REGION Network 4: AV-20.04
   RUNG wire#powerrail
      #"AV-20.04"(FB_OPEN := wire#w1, FB_CLOSE := wire#w2, LOCK := #lock, ERR_EXTERN :=, LIOP_SEL := #Init, L_AUT := #Init, L_REMOTE := #Init, L_SIM :=, L_RESET := #Reset, AUT_OP :=, MAN_OP :=, SIM_OP :=, L_MON := #Init, MON_T :=, MON_T_CLOSE :=, INSTANCE := 'AV-20.04', RESTART :=, VISIBILITY :=, OPdwCmd :=, QdwState =>, QwState =>, QCLOSING =>, QCLOSE =>, QOPENING =>, QOPEN =>, QCMD_OP => "AV-20.04", QMON =>, QMON_ERR =>, QMON_T =>, QMON_T_CLOSE =>, QMAN_AUT =>, QREMOTE =>, QSIM =>, QLOCK =>, QERR =>, QERR_EXT =>, QwAlarm =>)
   END_RUNG
   RUNG wire#powerrail
      Contact( #"AV-20.04".QCMD_OP )
   END_RUNG wire#w1
   RUNG wire#powerrail
      I_Contact( #"AV-20.04".QCMD_OP )
   END_RUNG wire#w2
   // the same network as SCL:
   #"AV-20.04"(LOCK := #lock,   // "Valve"
               LIOP_SEL := #Init,
               L_AUT := #Init,
               L_REMOTE := #Init,
               L_RESET := #Reset,
               FB_OPEN := #"AV-20.04".QCMD_OP,
               FB_CLOSE := NOT #"AV-20.04".QCMD_OP,
               L_MON := #Init,
               INSTANCE := 'AV-20.04',
               QCMD_OP => "AV-20.04");
END_REGION

REGION Network 5: AV-20.05
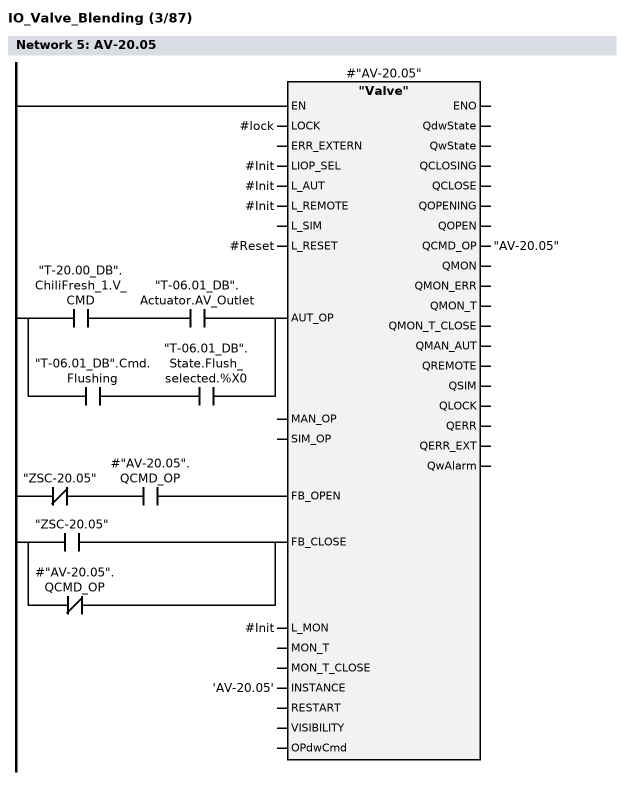
   RUNG wire#powerrail
      #"AV-20.05"(AUT_OP := wire#w1, FB_OPEN := wire#w2, FB_CLOSE := wire#w3, LOCK := #lock, ERR_EXTERN :=, LIOP_SEL := #Init, L_AUT := #Init, L_REMOTE := #Init, L_SIM :=, L_RESET := #Reset, MAN_OP :=, SIM_OP :=, L_MON := #Init, MON_T :=, MON_T_CLOSE :=, INSTANCE := 'AV-20.05', RESTART :=, VISIBILITY :=, OPdwCmd :=, QdwState =>, QwState =>, QCLOSING =>, QCLOSE =>, QOPENING =>, QOPEN =>, QCMD_OP => "AV-20.05", QMON =>, QMON_ERR =>, QMON_T =>, QMON_T_CLOSE =>, QMAN_AUT =>, QREMOTE =>, QSIM =>, QLOCK =>, QERR =>, QERR_EXT =>, QwAlarm =>)
   END_RUNG
   RUNG wire#powerrail
      Contact( "T-20.00_DB".ChiliFresh_1.V_CMD )
      Contact( "T-06.01_DB".Actuator.AV_Outlet )
   END_RUNG wire#w1
   RUNG wire#powerrail
      Contact( "T-06.01_DB".Cmd.Flushing )
      Contact( "T-06.01_DB".State.Flush_selected.%X0 )
   END_RUNG wire#w1
   RUNG wire#powerrail
      I_Contact( "ZSC-20.05" )
      Contact( #"AV-20.05".QCMD_OP )
   END_RUNG wire#w2
   RUNG wire#powerrail
      Contact( "ZSC-20.05" )
   END_RUNG wire#w3
   RUNG wire#powerrail
      I_Contact( #"AV-20.05".QCMD_OP )
   END_RUNG wire#w3
   // the same network as SCL:
   #"AV-20.05"(LOCK := #lock,   // "Valve"
               LIOP_SEL := #Init,
               L_AUT := #Init,
               L_REMOTE := #Init,
               L_RESET := #Reset,
               AUT_OP := ("T-20.00_DB".ChiliFresh_1.V_CMD AND "T-06.01_DB".Actuator.AV_Outlet) OR ("T-06.01_DB".Cmd.Flushing AND "T-06.01_DB".State.Flush_selected.%X0),
               FB_OPEN := NOT "ZSC-20.05" AND #"AV-20.05".QCMD_OP,
               FB_CLOSE := "ZSC-20.05" OR NOT #"AV-20.05".QCMD_OP,
               L_MON := #Init,
               INSTANCE := 'AV-20.05',
               QCMD_OP => "AV-20.05");
END_REGION

REGION Network 6: AV-20.06
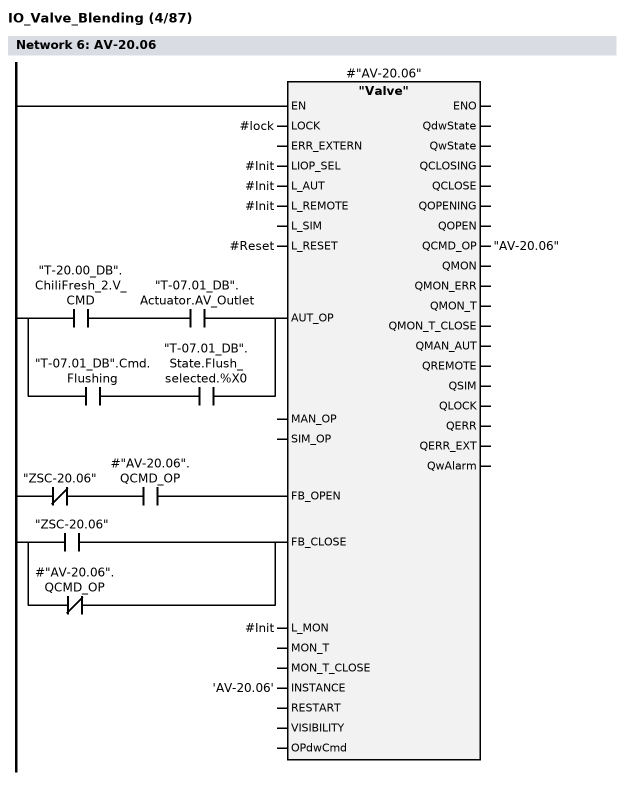
   RUNG wire#powerrail
      #"AV-20.06"(AUT_OP := wire#w1, FB_OPEN := wire#w2, FB_CLOSE := wire#w3, LOCK := #lock, ERR_EXTERN :=, LIOP_SEL := #Init, L_AUT := #Init, L_REMOTE := #Init, L_SIM :=, L_RESET := #Reset, MAN_OP :=, SIM_OP :=, L_MON := #Init, MON_T :=, MON_T_CLOSE :=, INSTANCE := 'AV-20.06', RESTART :=, VISIBILITY :=, OPdwCmd :=, QdwState =>, QwState =>, QCLOSING =>, QCLOSE =>, QOPENING =>, QOPEN =>, QCMD_OP => "AV-20.06", QMON =>, QMON_ERR =>, QMON_T =>, QMON_T_CLOSE =>, QMAN_AUT =>, QREMOTE =>, QSIM =>, QLOCK =>, QERR =>, QERR_EXT =>, QwAlarm =>)
   END_RUNG
   RUNG wire#powerrail
      Contact( "T-20.00_DB".ChiliFresh_2.V_CMD )
      Contact( "T-07.01_DB".Actuator.AV_Outlet )
   END_RUNG wire#w1
   RUNG wire#powerrail
      Contact( "T-07.01_DB".Cmd.Flushing )
      Contact( "T-07.01_DB".State.Flush_selected.%X0 )
   END_RUNG wire#w1
   RUNG wire#powerrail
      I_Contact( "ZSC-20.06" )
      Contact( #"AV-20.06".QCMD_OP )
   END_RUNG wire#w2
   RUNG wire#powerrail
      Contact( "ZSC-20.06" )
   END_RUNG wire#w3
   RUNG wire#powerrail
      I_Contact( #"AV-20.06".QCMD_OP )
   END_RUNG wire#w3
   // the same network as SCL:
   #"AV-20.06"(LOCK := #lock,   // "Valve"
               LIOP_SEL := #Init,
               L_AUT := #Init,
               L_REMOTE := #Init,
               L_RESET := #Reset,
               AUT_OP := ("T-20.00_DB".ChiliFresh_2.V_CMD AND "T-07.01_DB".Actuator.AV_Outlet) OR ("T-07.01_DB".Cmd.Flushing AND "T-07.01_DB".State.Flush_selected.%X0),
               FB_OPEN := NOT "ZSC-20.06" AND #"AV-20.06".QCMD_OP,
               FB_CLOSE := "ZSC-20.06" OR NOT #"AV-20.06".QCMD_OP,
               L_MON := #Init,
               INSTANCE := 'AV-20.06',
               QCMD_OP => "AV-20.06");
END_REGION

REGION Network 7: AV-20.07
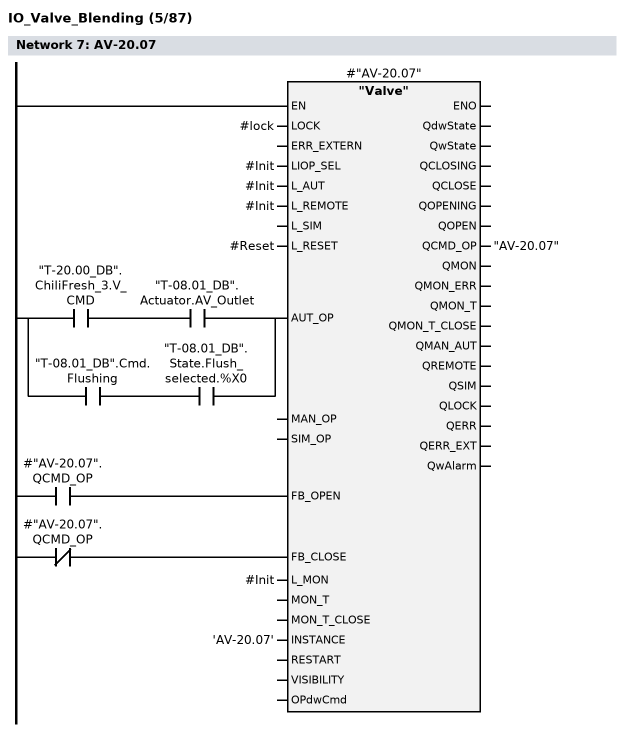
   RUNG wire#powerrail
      #"AV-20.07"(AUT_OP := wire#w1, FB_OPEN := wire#w2, FB_CLOSE := wire#w3, LOCK := #lock, ERR_EXTERN :=, LIOP_SEL := #Init, L_AUT := #Init, L_REMOTE := #Init, L_SIM :=, L_RESET := #Reset, MAN_OP :=, SIM_OP :=, L_MON := #Init, MON_T :=, MON_T_CLOSE :=, INSTANCE := 'AV-20.07', RESTART :=, VISIBILITY :=, OPdwCmd :=, QdwState =>, QwState =>, QCLOSING =>, QCLOSE =>, QOPENING =>, QOPEN =>, QCMD_OP => "AV-20.07", QMON =>, QMON_ERR =>, QMON_T =>, QMON_T_CLOSE =>, QMAN_AUT =>, QREMOTE =>, QSIM =>, QLOCK =>, QERR =>, QERR_EXT =>, QwAlarm =>)
   END_RUNG
   RUNG wire#powerrail
      Contact( "T-20.00_DB".ChiliFresh_3.V_CMD )
      Contact( "T-08.01_DB".Actuator.AV_Outlet )
   END_RUNG wire#w1
   RUNG wire#powerrail
      Contact( "T-08.01_DB".Cmd.Flushing )
      Contact( "T-08.01_DB".State.Flush_selected.%X0 )
   END_RUNG wire#w1
   RUNG wire#powerrail
      Contact( #"AV-20.07".QCMD_OP )
   END_RUNG wire#w2
   RUNG wire#powerrail
      I_Contact( #"AV-20.07".QCMD_OP )
   END_RUNG wire#w3
   // the same network as SCL:
   #"AV-20.07"(LOCK := #lock,   // "Valve"
               LIOP_SEL := #Init,
               L_AUT := #Init,
               L_REMOTE := #Init,
               L_RESET := #Reset,
               AUT_OP := ("T-20.00_DB".ChiliFresh_3.V_CMD AND "T-08.01_DB".Actuator.AV_Outlet) OR ("T-08.01_DB".Cmd.Flushing AND "T-08.01_DB".State.Flush_selected.%X0),
               FB_OPEN := #"AV-20.07".QCMD_OP,
               FB_CLOSE := NOT #"AV-20.07".QCMD_OP,
               L_MON := #Init,
               INSTANCE := 'AV-20.07',
               QCMD_OP => "AV-20.07");
END_REGION

REGION Network 8: AV-20.08
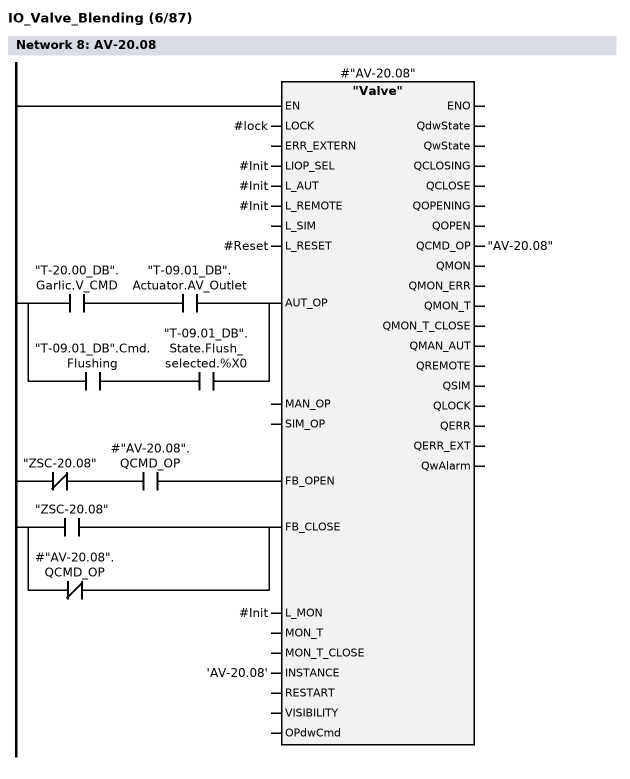
   RUNG wire#powerrail
      #"AV-20.08"(AUT_OP := wire#w1, FB_OPEN := wire#w2, FB_CLOSE := wire#w3, LOCK := #lock, ERR_EXTERN :=, LIOP_SEL := #Init, L_AUT := #Init, L_REMOTE := #Init, L_SIM :=, L_RESET := #Reset, MAN_OP :=, SIM_OP :=, L_MON := #Init, MON_T :=, MON_T_CLOSE :=, INSTANCE := 'AV-20.08', RESTART :=, VISIBILITY :=, OPdwCmd :=, QdwState =>, QwState =>, QCLOSING =>, QCLOSE =>, QOPENING =>, QOPEN =>, QCMD_OP => "AV-20.08", QMON =>, QMON_ERR =>, QMON_T =>, QMON_T_CLOSE =>, QMAN_AUT =>, QREMOTE =>, QSIM =>, QLOCK =>, QERR =>, QERR_EXT =>, QwAlarm =>)
   END_RUNG
   RUNG wire#powerrail
      Contact( "T-20.00_DB".Garlic.V_CMD )
      Contact( "T-09.01_DB".Actuator.AV_Outlet )
   END_RUNG wire#w1
   RUNG wire#powerrail
      Contact( "T-09.01_DB".Cmd.Flushing )
      Contact( "T-09.01_DB".State.Flush_selected.%X0 )
   END_RUNG wire#w1
   RUNG wire#powerrail
      I_Contact( "ZSC-20.08" )
      Contact( #"AV-20.08".QCMD_OP )
   END_RUNG wire#w2
   RUNG wire#powerrail
      Contact( "ZSC-20.08" )
   END_RUNG wire#w3
   RUNG wire#powerrail
      I_Contact( #"AV-20.08".QCMD_OP )
   END_RUNG wire#w3
   // the same network as SCL:
   #"AV-20.08"(LOCK := #lock,   // "Valve"
               LIOP_SEL := #Init,
               L_AUT := #Init,
               L_REMOTE := #Init,
               L_RESET := #Reset,
               AUT_OP := ("T-20.00_DB".Garlic.V_CMD AND "T-09.01_DB".Actuator.AV_Outlet) OR ("T-09.01_DB".Cmd.Flushing AND "T-09.01_DB".State.Flush_selected.%X0),
               FB_OPEN := NOT "ZSC-20.08" AND #"AV-20.08".QCMD_OP,
               FB_CLOSE := "ZSC-20.08" OR NOT #"AV-20.08".QCMD_OP,
               L_MON := #Init,
               INSTANCE := 'AV-20.08',
               QCMD_OP => "AV-20.08");
END_REGION

REGION Network 9: AV-20.09
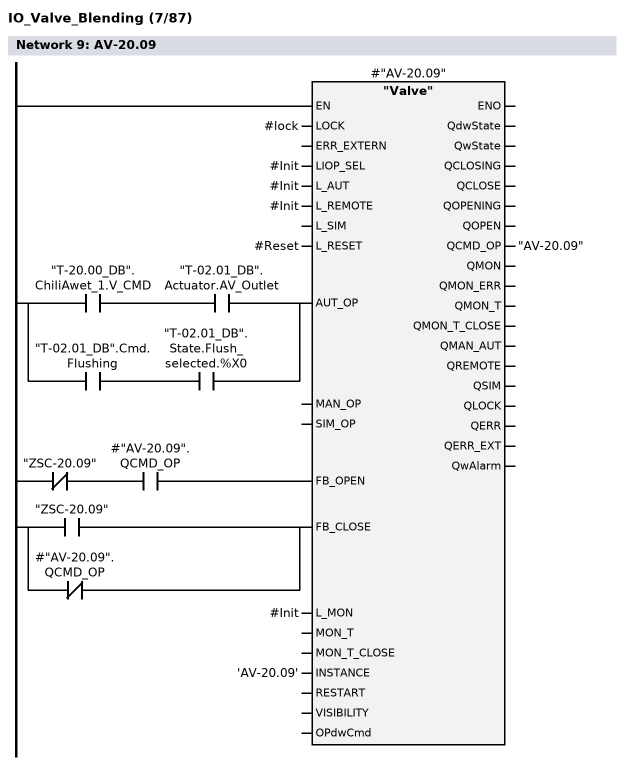
   RUNG wire#powerrail
      #"AV-20.09"(AUT_OP := wire#w1, FB_OPEN := wire#w2, FB_CLOSE := wire#w3, LOCK := #lock, ERR_EXTERN :=, LIOP_SEL := #Init, L_AUT := #Init, L_REMOTE := #Init, L_SIM :=, L_RESET := #Reset, MAN_OP :=, SIM_OP :=, L_MON := #Init, MON_T :=, MON_T_CLOSE :=, INSTANCE := 'AV-20.09', RESTART :=, VISIBILITY :=, OPdwCmd :=, QdwState =>, QwState =>, QCLOSING =>, QCLOSE =>, QOPENING =>, QOPEN =>, QCMD_OP => "AV-20.09", QMON =>, QMON_ERR =>, QMON_T =>, QMON_T_CLOSE =>, QMAN_AUT =>, QREMOTE =>, QSIM =>, QLOCK =>, QERR =>, QERR_EXT =>, QwAlarm =>)
   END_RUNG
   RUNG wire#powerrail
      Contact( "T-20.00_DB".ChiliAwet_1.V_CMD )
      Contact( "T-02.01_DB".Actuator.AV_Outlet )
   END_RUNG wire#w1
   RUNG wire#powerrail
      Contact( "T-02.01_DB".Cmd.Flushing )
      Contact( "T-02.01_DB".State.Flush_selected.%X0 )
   END_RUNG wire#w1
   RUNG wire#powerrail
      I_Contact( "ZSC-20.09" )
      Contact( #"AV-20.09".QCMD_OP )
   END_RUNG wire#w2
   RUNG wire#powerrail
      Contact( "ZSC-20.09" )
   END_RUNG wire#w3
   RUNG wire#powerrail
      I_Contact( #"AV-20.09".QCMD_OP )
   END_RUNG wire#w3
   // the same network as SCL:
   #"AV-20.09"(LOCK := #lock,   // "Valve"
               LIOP_SEL := #Init,
               L_AUT := #Init,
               L_REMOTE := #Init,
               L_RESET := #Reset,
               AUT_OP := ("T-20.00_DB".ChiliAwet_1.V_CMD AND "T-02.01_DB".Actuator.AV_Outlet) OR ("T-02.01_DB".Cmd.Flushing AND "T-02.01_DB".State.Flush_selected.%X0),
               FB_OPEN := NOT "ZSC-20.09" AND #"AV-20.09".QCMD_OP,
               FB_CLOSE := "ZSC-20.09" OR NOT #"AV-20.09".QCMD_OP,
               L_MON := #Init,
               INSTANCE := 'AV-20.09',
               QCMD_OP => "AV-20.09");
END_REGION

REGION Network 10: AV-20.10
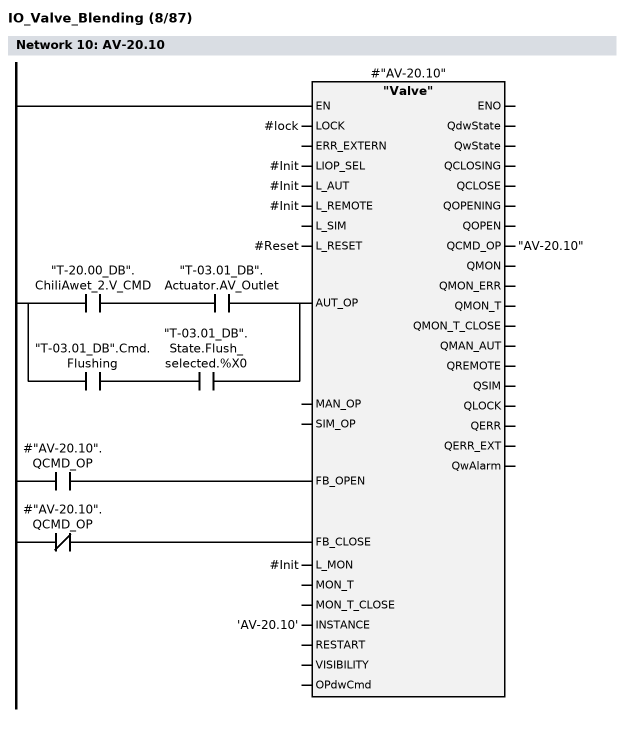
   RUNG wire#powerrail
      #"AV-20.10"(AUT_OP := wire#w1, FB_OPEN := wire#w2, FB_CLOSE := wire#w3, LOCK := #lock, ERR_EXTERN :=, LIOP_SEL := #Init, L_AUT := #Init, L_REMOTE := #Init, L_SIM :=, L_RESET := #Reset, MAN_OP :=, SIM_OP :=, L_MON := #Init, MON_T :=, MON_T_CLOSE :=, INSTANCE := 'AV-20.10', RESTART :=, VISIBILITY :=, OPdwCmd :=, QdwState =>, QwState =>, QCLOSING =>, QCLOSE =>, QOPENING =>, QOPEN =>, QCMD_OP => "AV-20.10", QMON =>, QMON_ERR =>, QMON_T =>, QMON_T_CLOSE =>, QMAN_AUT =>, QREMOTE =>, QSIM =>, QLOCK =>, QERR =>, QERR_EXT =>, QwAlarm =>)
   END_RUNG
   RUNG wire#powerrail
      Contact( "T-20.00_DB".ChiliAwet_2.V_CMD )
      Contact( "T-03.01_DB".Actuator.AV_Outlet )
   END_RUNG wire#w1
   RUNG wire#powerrail
      Contact( "T-03.01_DB".Cmd.Flushing )
      Contact( "T-03.01_DB".State.Flush_selected.%X0 )
   END_RUNG wire#w1
   RUNG wire#powerrail
      Contact( #"AV-20.10".QCMD_OP )
   END_RUNG wire#w2
   RUNG wire#powerrail
      I_Contact( #"AV-20.10".QCMD_OP )
   END_RUNG wire#w3
   // the same network as SCL:
   #"AV-20.10"(LOCK := #lock,   // "Valve"
               LIOP_SEL := #Init,
               L_AUT := #Init,
               L_REMOTE := #Init,
               L_RESET := #Reset,
               AUT_OP := ("T-20.00_DB".ChiliAwet_2.V_CMD AND "T-03.01_DB".Actuator.AV_Outlet) OR ("T-03.01_DB".Cmd.Flushing AND "T-03.01_DB".State.Flush_selected.%X0),
               FB_OPEN := #"AV-20.10".QCMD_OP,
               FB_CLOSE := NOT #"AV-20.10".QCMD_OP,
               L_MON := #Init,
               INSTANCE := 'AV-20.10',
               QCMD_OP => "AV-20.10");
END_REGION

REGION Network 11: AV-20.11
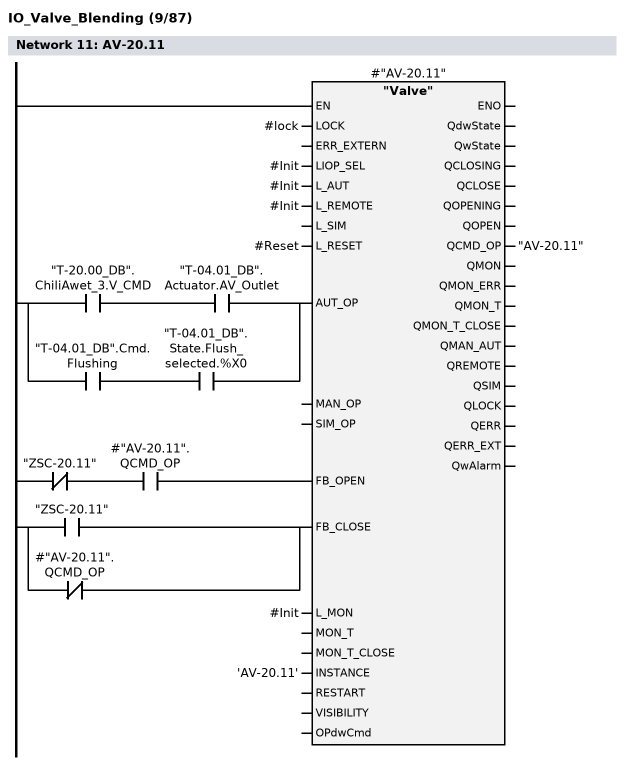
   RUNG wire#powerrail
      #"AV-20.11"(AUT_OP := wire#w1, FB_OPEN := wire#w2, FB_CLOSE := wire#w3, LOCK := #lock, ERR_EXTERN :=, LIOP_SEL := #Init, L_AUT := #Init, L_REMOTE := #Init, L_SIM :=, L_RESET := #Reset, MAN_OP :=, SIM_OP :=, L_MON := #Init, MON_T :=, MON_T_CLOSE :=, INSTANCE := 'AV-20.11', RESTART :=, VISIBILITY :=, OPdwCmd :=, QdwState =>, QwState =>, QCLOSING =>, QCLOSE =>, QOPENING =>, QOPEN =>, QCMD_OP => "AV-20.11", QMON =>, QMON_ERR =>, QMON_T =>, QMON_T_CLOSE =>, QMAN_AUT =>, QREMOTE =>, QSIM =>, QLOCK =>, QERR =>, QERR_EXT =>, QwAlarm =>)
   END_RUNG
   RUNG wire#powerrail
      Contact( "T-20.00_DB".ChiliAwet_3.V_CMD )
      Contact( "T-04.01_DB".Actuator.AV_Outlet )
   END_RUNG wire#w1
   RUNG wire#powerrail
      Contact( "T-04.01_DB".Cmd.Flushing )
      Contact( "T-04.01_DB".State.Flush_selected.%X0 )
   END_RUNG wire#w1
   RUNG wire#powerrail
      I_Contact( "ZSC-20.11" )
      Contact( #"AV-20.11".QCMD_OP )
   END_RUNG wire#w2
   RUNG wire#powerrail
      Contact( "ZSC-20.11" )
   END_RUNG wire#w3
   RUNG wire#powerrail
      I_Contact( #"AV-20.11".QCMD_OP )
   END_RUNG wire#w3
   // the same network as SCL:
   #"AV-20.11"(LOCK := #lock,   // "Valve"
               LIOP_SEL := #Init,
               L_AUT := #Init,
               L_REMOTE := #Init,
               L_RESET := #Reset,
               AUT_OP := ("T-20.00_DB".ChiliAwet_3.V_CMD AND "T-04.01_DB".Actuator.AV_Outlet) OR ("T-04.01_DB".Cmd.Flushing AND "T-04.01_DB".State.Flush_selected.%X0),
               FB_OPEN := NOT "ZSC-20.11" AND #"AV-20.11".QCMD_OP,
               FB_CLOSE := "ZSC-20.11" OR NOT #"AV-20.11".QCMD_OP,
               L_MON := #Init,
               INSTANCE := 'AV-20.11',
               QCMD_OP => "AV-20.11");
END_REGION

REGION Network 12: AV-20.12
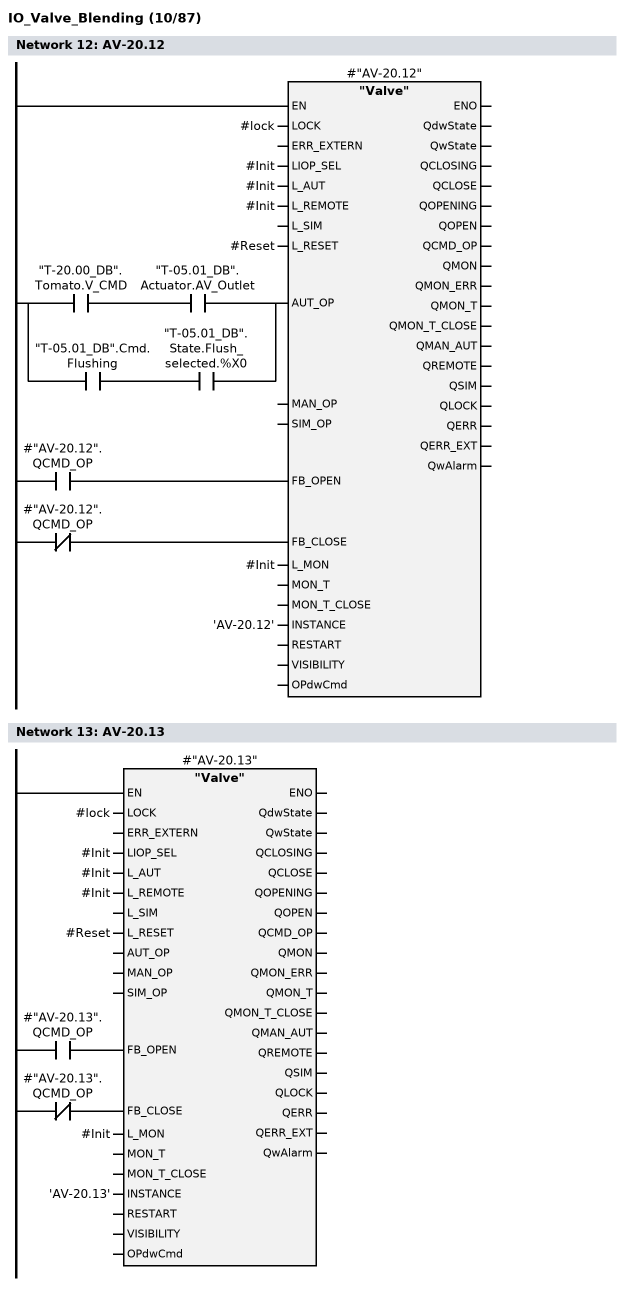
   RUNG wire#powerrail
      #"AV-20.12"(AUT_OP := wire#w1, FB_OPEN := wire#w2, FB_CLOSE := wire#w3, LOCK := #lock, ERR_EXTERN :=, LIOP_SEL := #Init, L_AUT := #Init, L_REMOTE := #Init, L_SIM :=, L_RESET := #Reset, MAN_OP :=, SIM_OP :=, L_MON := #Init, MON_T :=, MON_T_CLOSE :=, INSTANCE := 'AV-20.12', RESTART :=, VISIBILITY :=, OPdwCmd :=, QdwState =>, QwState =>, QCLOSING =>, QCLOSE =>, QOPENING =>, QOPEN =>, QCMD_OP =>, QMON =>, QMON_ERR =>, QMON_T =>, QMON_T_CLOSE =>, QMAN_AUT =>, QREMOTE =>, QSIM =>, QLOCK =>, QERR =>, QERR_EXT =>, QwAlarm =>)
   END_RUNG
   RUNG wire#powerrail
      Contact( "T-20.00_DB".Tomato.V_CMD )
      Contact( "T-05.01_DB".Actuator.AV_Outlet )
   END_RUNG wire#w1
   RUNG wire#powerrail
      Contact( "T-05.01_DB".Cmd.Flushing )
      Contact( "T-05.01_DB".State.Flush_selected.%X0 )
   END_RUNG wire#w1
   RUNG wire#powerrail
      Contact( #"AV-20.12".QCMD_OP )
   END_RUNG wire#w2
   RUNG wire#powerrail
      I_Contact( #"AV-20.12".QCMD_OP )
   END_RUNG wire#w3
   // the same network as SCL:
   #"AV-20.12"(LOCK := #lock,   // "Valve"
               LIOP_SEL := #Init,
               L_AUT := #Init,
               L_REMOTE := #Init,
               L_RESET := #Reset,
               AUT_OP := ("T-20.00_DB".Tomato.V_CMD AND "T-05.01_DB".Actuator.AV_Outlet) OR ("T-05.01_DB".Cmd.Flushing AND "T-05.01_DB".State.Flush_selected.%X0),
               FB_OPEN := #"AV-20.12".QCMD_OP,
               FB_CLOSE := NOT #"AV-20.12".QCMD_OP,
               L_MON := #Init,
               INSTANCE := 'AV-20.12');
END_REGION

REGION Network 13: AV-20.13
   RUNG wire#powerrail
      #"AV-20.13"(FB_OPEN := wire#w1, FB_CLOSE := wire#w2, LOCK := #lock, ERR_EXTERN :=, LIOP_SEL := #Init, L_AUT := #Init, L_REMOTE := #Init, L_SIM :=, L_RESET := #Reset, AUT_OP :=, MAN_OP :=, SIM_OP :=, L_MON := #Init, MON_T :=, MON_T_CLOSE :=, INSTANCE := 'AV-20.13', RESTART :=, VISIBILITY :=, OPdwCmd :=, QdwState =>, QwState =>, QCLOSING =>, QCLOSE =>, QOPENING =>, QOPEN =>, QCMD_OP =>, QMON =>, QMON_ERR =>, QMON_T =>, QMON_T_CLOSE =>, QMAN_AUT =>, QREMOTE =>, QSIM =>, QLOCK =>, QERR =>, QERR_EXT =>, QwAlarm =>)
   END_RUNG
   RUNG wire#powerrail
      Contact( #"AV-20.13".QCMD_OP )
   END_RUNG wire#w1
   RUNG wire#powerrail
      I_Contact( #"AV-20.13".QCMD_OP )
   END_RUNG wire#w2
   // the same network as SCL:
   #"AV-20.13"(LOCK := #lock,   // "Valve"
               LIOP_SEL := #Init,
               L_AUT := #Init,
               L_REMOTE := #Init,
               L_RESET := #Reset,
               FB_OPEN := #"AV-20.13".QCMD_OP,
               FB_CLOSE := NOT #"AV-20.13".QCMD_OP,
               L_MON := #Init,
               INSTANCE := 'AV-20.13');
END_REGION

REGION Network 14: AV-20.14
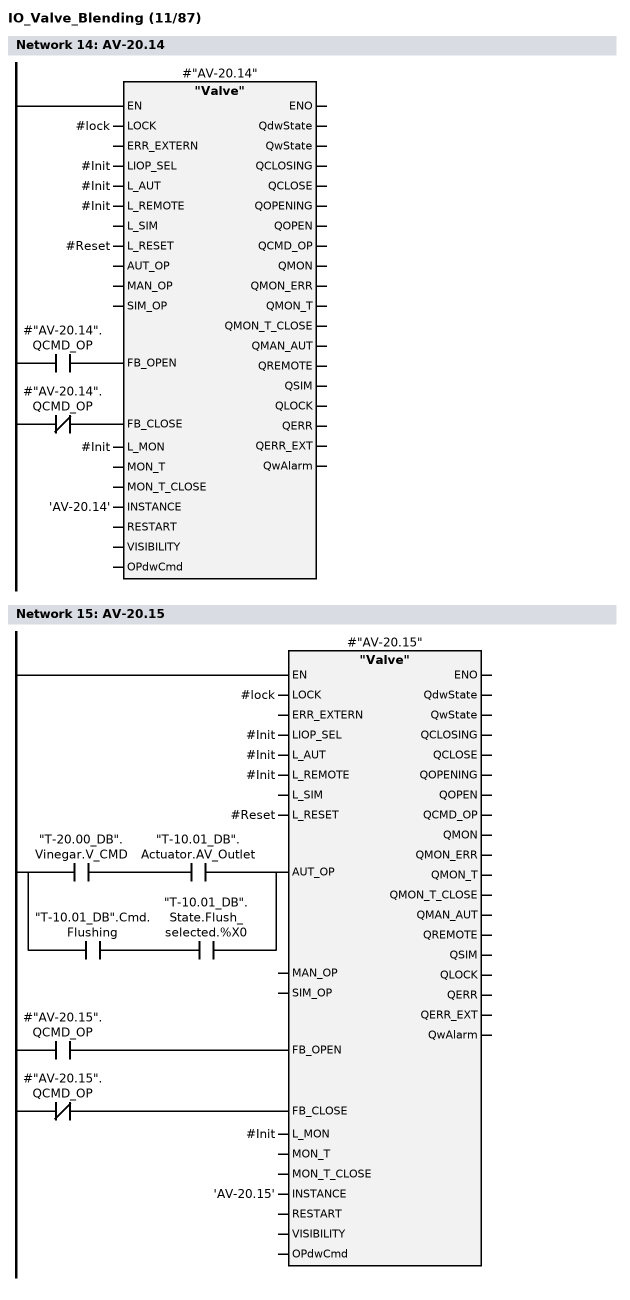
   RUNG wire#powerrail
      #"AV-20.14"(FB_OPEN := wire#w1, FB_CLOSE := wire#w2, LOCK := #lock, ERR_EXTERN :=, LIOP_SEL := #Init, L_AUT := #Init, L_REMOTE := #Init, L_SIM :=, L_RESET := #Reset, AUT_OP :=, MAN_OP :=, SIM_OP :=, L_MON := #Init, MON_T :=, MON_T_CLOSE :=, INSTANCE := 'AV-20.14', RESTART :=, VISIBILITY :=, OPdwCmd :=, QdwState =>, QwState =>, QCLOSING =>, QCLOSE =>, QOPENING =>, QOPEN =>, QCMD_OP =>, QMON =>, QMON_ERR =>, QMON_T =>, QMON_T_CLOSE =>, QMAN_AUT =>, QREMOTE =>, QSIM =>, QLOCK =>, QERR =>, QERR_EXT =>, QwAlarm =>)
   END_RUNG
   RUNG wire#powerrail
      Contact( #"AV-20.14".QCMD_OP )
   END_RUNG wire#w1
   RUNG wire#powerrail
      I_Contact( #"AV-20.14".QCMD_OP )
   END_RUNG wire#w2
   // the same network as SCL:
   #"AV-20.14"(LOCK := #lock,   // "Valve"
               LIOP_SEL := #Init,
               L_AUT := #Init,
               L_REMOTE := #Init,
               L_RESET := #Reset,
               FB_OPEN := #"AV-20.14".QCMD_OP,
               FB_CLOSE := NOT #"AV-20.14".QCMD_OP,
               L_MON := #Init,
               INSTANCE := 'AV-20.14');
END_REGION

REGION Network 15: AV-20.15
   RUNG wire#powerrail
      #"AV-20.15"(AUT_OP := wire#w1, FB_OPEN := wire#w2, FB_CLOSE := wire#w3, LOCK := #lock, ERR_EXTERN :=, LIOP_SEL := #Init, L_AUT := #Init, L_REMOTE := #Init, L_SIM :=, L_RESET := #Reset, MAN_OP :=, SIM_OP :=, L_MON := #Init, MON_T :=, MON_T_CLOSE :=, INSTANCE := 'AV-20.15', RESTART :=, VISIBILITY :=, OPdwCmd :=, QdwState =>, QwState =>, QCLOSING =>, QCLOSE =>, QOPENING =>, QOPEN =>, QCMD_OP =>, QMON =>, QMON_ERR =>, QMON_T =>, QMON_T_CLOSE =>, QMAN_AUT =>, QREMOTE =>, QSIM =>, QLOCK =>, QERR =>, QERR_EXT =>, QwAlarm =>)
   END_RUNG
   RUNG wire#powerrail
      Contact( "T-20.00_DB".Vinegar.V_CMD )
      Contact( "T-10.01_DB".Actuator.AV_Outlet )
   END_RUNG wire#w1
   RUNG wire#powerrail
      Contact( "T-10.01_DB".Cmd.Flushing )
      Contact( "T-10.01_DB".State.Flush_selected.%X0 )
   END_RUNG wire#w1
   RUNG wire#powerrail
      Contact( #"AV-20.15".QCMD_OP )
   END_RUNG wire#w2
   RUNG wire#powerrail
      I_Contact( #"AV-20.15".QCMD_OP )
   END_RUNG wire#w3
   // the same network as SCL:
   #"AV-20.15"(LOCK := #lock,   // "Valve"
               LIOP_SEL := #Init,
               L_AUT := #Init,
               L_REMOTE := #Init,
               L_RESET := #Reset,
               AUT_OP := ("T-20.00_DB".Vinegar.V_CMD AND "T-10.01_DB".Actuator.AV_Outlet) OR ("T-10.01_DB".Cmd.Flushing AND "T-10.01_DB".State.Flush_selected.%X0),
               FB_OPEN := #"AV-20.15".QCMD_OP,
               FB_CLOSE := NOT #"AV-20.15".QCMD_OP,
               L_MON := #Init,
               INSTANCE := 'AV-20.15');
END_REGION

REGION Network 16: AV-20.16
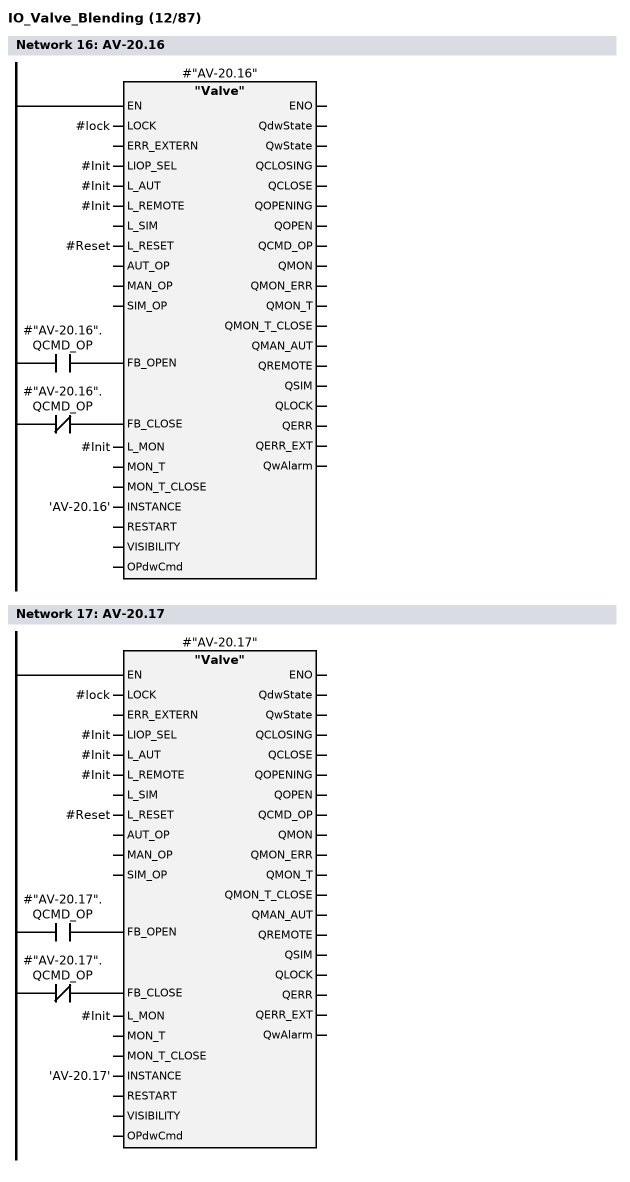
   RUNG wire#powerrail
      #"AV-20.16"(FB_OPEN := wire#w1, FB_CLOSE := wire#w2, LOCK := #lock, ERR_EXTERN :=, LIOP_SEL := #Init, L_AUT := #Init, L_REMOTE := #Init, L_SIM :=, L_RESET := #Reset, AUT_OP :=, MAN_OP :=, SIM_OP :=, L_MON := #Init, MON_T :=, MON_T_CLOSE :=, INSTANCE := 'AV-20.16', RESTART :=, VISIBILITY :=, OPdwCmd :=, QdwState =>, QwState =>, QCLOSING =>, QCLOSE =>, QOPENING =>, QOPEN =>, QCMD_OP =>, QMON =>, QMON_ERR =>, QMON_T =>, QMON_T_CLOSE =>, QMAN_AUT =>, QREMOTE =>, QSIM =>, QLOCK =>, QERR =>, QERR_EXT =>, QwAlarm =>)
   END_RUNG
   RUNG wire#powerrail
      Contact( #"AV-20.16".QCMD_OP )
   END_RUNG wire#w1
   RUNG wire#powerrail
      I_Contact( #"AV-20.16".QCMD_OP )
   END_RUNG wire#w2
   // the same network as SCL:
   #"AV-20.16"(LOCK := #lock,   // "Valve"
               LIOP_SEL := #Init,
               L_AUT := #Init,
               L_REMOTE := #Init,
               L_RESET := #Reset,
               FB_OPEN := #"AV-20.16".QCMD_OP,
               FB_CLOSE := NOT #"AV-20.16".QCMD_OP,
               L_MON := #Init,
               INSTANCE := 'AV-20.16');
END_REGION

REGION Network 17: AV-20.17
   RUNG wire#powerrail
      #"AV-20.17"(FB_OPEN := wire#w1, FB_CLOSE := wire#w2, LOCK := #lock, ERR_EXTERN :=, LIOP_SEL := #Init, L_AUT := #Init, L_REMOTE := #Init, L_SIM :=, L_RESET := #Reset, AUT_OP :=, MAN_OP :=, SIM_OP :=, L_MON := #Init, MON_T :=, MON_T_CLOSE :=, INSTANCE := 'AV-20.17', RESTART :=, VISIBILITY :=, OPdwCmd :=, QdwState =>, QwState =>, QCLOSING =>, QCLOSE =>, QOPENING =>, QOPEN =>, QCMD_OP =>, QMON =>, QMON_ERR =>, QMON_T =>, QMON_T_CLOSE =>, QMAN_AUT =>, QREMOTE =>, QSIM =>, QLOCK =>, QERR =>, QERR_EXT =>, QwAlarm =>)
   END_RUNG
   RUNG wire#powerrail
      Contact( #"AV-20.17".QCMD_OP )
   END_RUNG wire#w1
   RUNG wire#powerrail
      I_Contact( #"AV-20.17".QCMD_OP )
   END_RUNG wire#w2
   // the same network as SCL:
   #"AV-20.17"(LOCK := #lock,   // "Valve"
               LIOP_SEL := #Init,
               L_AUT := #Init,
               L_REMOTE := #Init,
               L_RESET := #Reset,
               FB_OPEN := #"AV-20.17".QCMD_OP,
               FB_CLOSE := NOT #"AV-20.17".QCMD_OP,
               L_MON := #Init,
               INSTANCE := 'AV-20.17');
END_REGION

REGION Network 18: AV-20.31
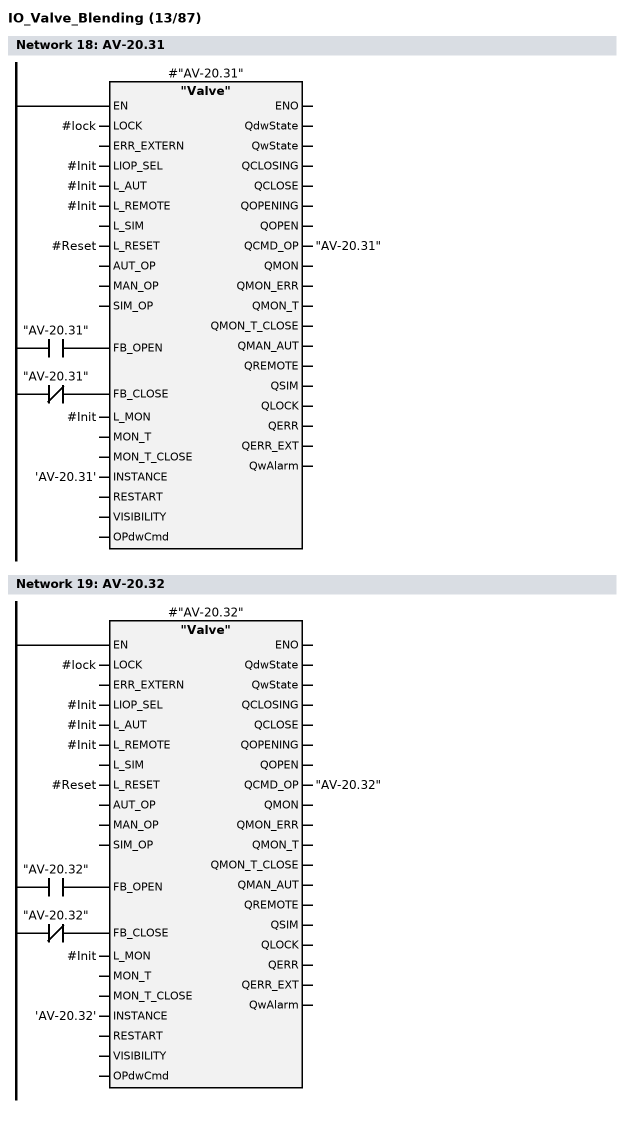
   RUNG wire#powerrail
      #"AV-20.31"(FB_OPEN := wire#w1, FB_CLOSE := wire#w2, LOCK := #lock, ERR_EXTERN :=, LIOP_SEL := #Init, L_AUT := #Init, L_REMOTE := #Init, L_SIM :=, L_RESET := #Reset, AUT_OP :=, MAN_OP :=, SIM_OP :=, L_MON := #Init, MON_T :=, MON_T_CLOSE :=, INSTANCE := 'AV-20.31', RESTART :=, VISIBILITY :=, OPdwCmd :=, QdwState =>, QwState =>, QCLOSING =>, QCLOSE =>, QOPENING =>, QOPEN =>, QCMD_OP => "AV-20.31", QMON =>, QMON_ERR =>, QMON_T =>, QMON_T_CLOSE =>, QMAN_AUT =>, QREMOTE =>, QSIM =>, QLOCK =>, QERR =>, QERR_EXT =>, QwAlarm =>)
   END_RUNG
   RUNG wire#powerrail
      Contact( "AV-20.31" )
   END_RUNG wire#w1
   RUNG wire#powerrail
      I_Contact( "AV-20.31" )
   END_RUNG wire#w2
   // the same network as SCL:
   #"AV-20.31"(LOCK := #lock,   // "Valve"
               LIOP_SEL := #Init,
               L_AUT := #Init,
               L_REMOTE := #Init,
               L_RESET := #Reset,
               FB_OPEN := "AV-20.31",
               FB_CLOSE := NOT "AV-20.31",
               L_MON := #Init,
               INSTANCE := 'AV-20.31',
               QCMD_OP => "AV-20.31");
END_REGION

REGION Network 19: AV-20.32
   RUNG wire#powerrail
      #"AV-20.32"(FB_OPEN := wire#w1, FB_CLOSE := wire#w2, LOCK := #lock, ERR_EXTERN :=, LIOP_SEL := #Init, L_AUT := #Init, L_REMOTE := #Init, L_SIM :=, L_RESET := #Reset, AUT_OP :=, MAN_OP :=, SIM_OP :=, L_MON := #Init, MON_T :=, MON_T_CLOSE :=, INSTANCE := 'AV-20.32', RESTART :=, VISIBILITY :=, OPdwCmd :=, QdwState =>, QwState =>, QCLOSING =>, QCLOSE =>, QOPENING =>, QOPEN =>, QCMD_OP => "AV-20.32", QMON =>, QMON_ERR =>, QMON_T =>, QMON_T_CLOSE =>, QMAN_AUT =>, QREMOTE =>, QSIM =>, QLOCK =>, QERR =>, QERR_EXT =>, QwAlarm =>)
   END_RUNG
   RUNG wire#powerrail
      Contact( "AV-20.32" )
   END_RUNG wire#w1
   RUNG wire#powerrail
      I_Contact( "AV-20.32" )
   END_RUNG wire#w2
   // the same network as SCL:
   #"AV-20.32"(LOCK := #lock,   // "Valve"
               LIOP_SEL := #Init,
               L_AUT := #Init,
               L_REMOTE := #Init,
               L_RESET := #Reset,
               FB_OPEN := "AV-20.32",
               FB_CLOSE := NOT "AV-20.32",
               L_MON := #Init,
               INSTANCE := 'AV-20.32',
               QCMD_OP => "AV-20.32");
END_REGION

REGION Network 20: AV-20.33
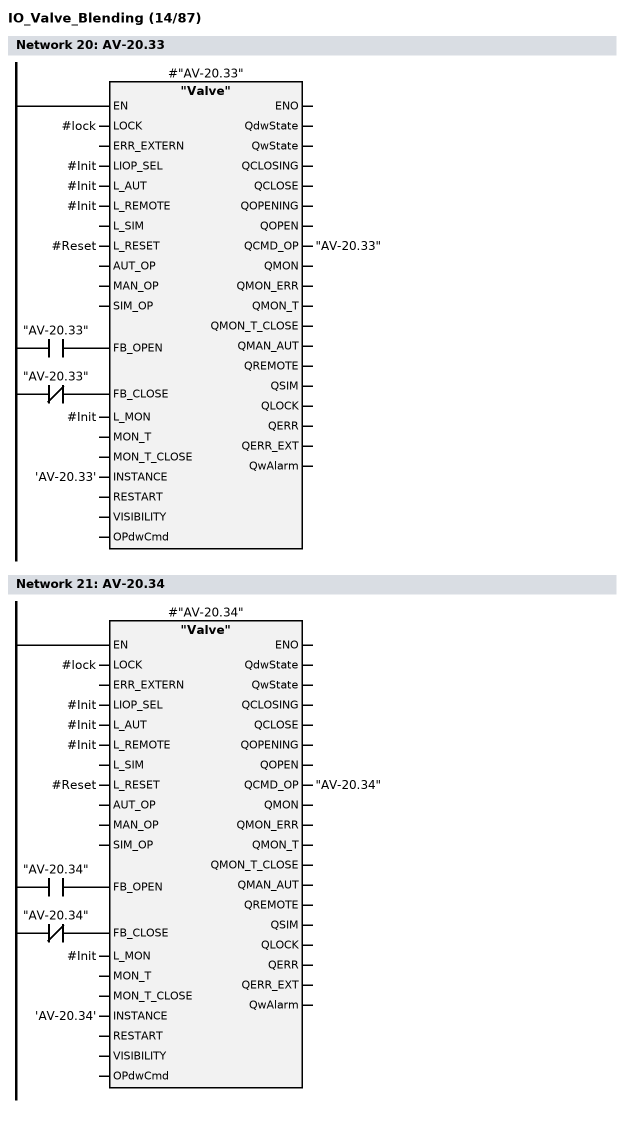
   RUNG wire#powerrail
      #"AV-20.33"(FB_OPEN := wire#w1, FB_CLOSE := wire#w2, LOCK := #lock, ERR_EXTERN :=, LIOP_SEL := #Init, L_AUT := #Init, L_REMOTE := #Init, L_SIM :=, L_RESET := #Reset, AUT_OP :=, MAN_OP :=, SIM_OP :=, L_MON := #Init, MON_T :=, MON_T_CLOSE :=, INSTANCE := 'AV-20.33', RESTART :=, VISIBILITY :=, OPdwCmd :=, QdwState =>, QwState =>, QCLOSING =>, QCLOSE =>, QOPENING =>, QOPEN =>, QCMD_OP => "AV-20.33", QMON =>, QMON_ERR =>, QMON_T =>, QMON_T_CLOSE =>, QMAN_AUT =>, QREMOTE =>, QSIM =>, QLOCK =>, QERR =>, QERR_EXT =>, QwAlarm =>)
   END_RUNG
   RUNG wire#powerrail
      Contact( "AV-20.33" )
   END_RUNG wire#w1
   RUNG wire#powerrail
      I_Contact( "AV-20.33" )
   END_RUNG wire#w2
   // the same network as SCL:
   #"AV-20.33"(LOCK := #lock,   // "Valve"
               LIOP_SEL := #Init,
               L_AUT := #Init,
               L_REMOTE := #Init,
               L_RESET := #Reset,
               FB_OPEN := "AV-20.33",
               FB_CLOSE := NOT "AV-20.33",
               L_MON := #Init,
               INSTANCE := 'AV-20.33',
               QCMD_OP => "AV-20.33");
END_REGION

REGION Network 21: AV-20.34
   RUNG wire#powerrail
      #"AV-20.34"(FB_OPEN := wire#w1, FB_CLOSE := wire#w2, LOCK := #lock, ERR_EXTERN :=, LIOP_SEL := #Init, L_AUT := #Init, L_REMOTE := #Init, L_SIM :=, L_RESET := #Reset, AUT_OP :=, MAN_OP :=, SIM_OP :=, L_MON := #Init, MON_T :=, MON_T_CLOSE :=, INSTANCE := 'AV-20.34', RESTART :=, VISIBILITY :=, OPdwCmd :=, QdwState =>, QwState =>, QCLOSING =>, QCLOSE =>, QOPENING =>, QOPEN =>, QCMD_OP => "AV-20.34", QMON =>, QMON_ERR =>, QMON_T =>, QMON_T_CLOSE =>, QMAN_AUT =>, QREMOTE =>, QSIM =>, QLOCK =>, QERR =>, QERR_EXT =>, QwAlarm =>)
   END_RUNG
   RUNG wire#powerrail
      Contact( "AV-20.34" )
   END_RUNG wire#w1
   RUNG wire#powerrail
      I_Contact( "AV-20.34" )
   END_RUNG wire#w2
   // the same network as SCL:
   #"AV-20.34"(LOCK := #lock,   // "Valve"
               LIOP_SEL := #Init,
               L_AUT := #Init,
               L_REMOTE := #Init,
               L_RESET := #Reset,
               FB_OPEN := "AV-20.34",
               FB_CLOSE := NOT "AV-20.34",
               L_MON := #Init,
               INSTANCE := 'AV-20.34',
               QCMD_OP => "AV-20.34");
END_REGION

REGION Network 22: AV-20.35
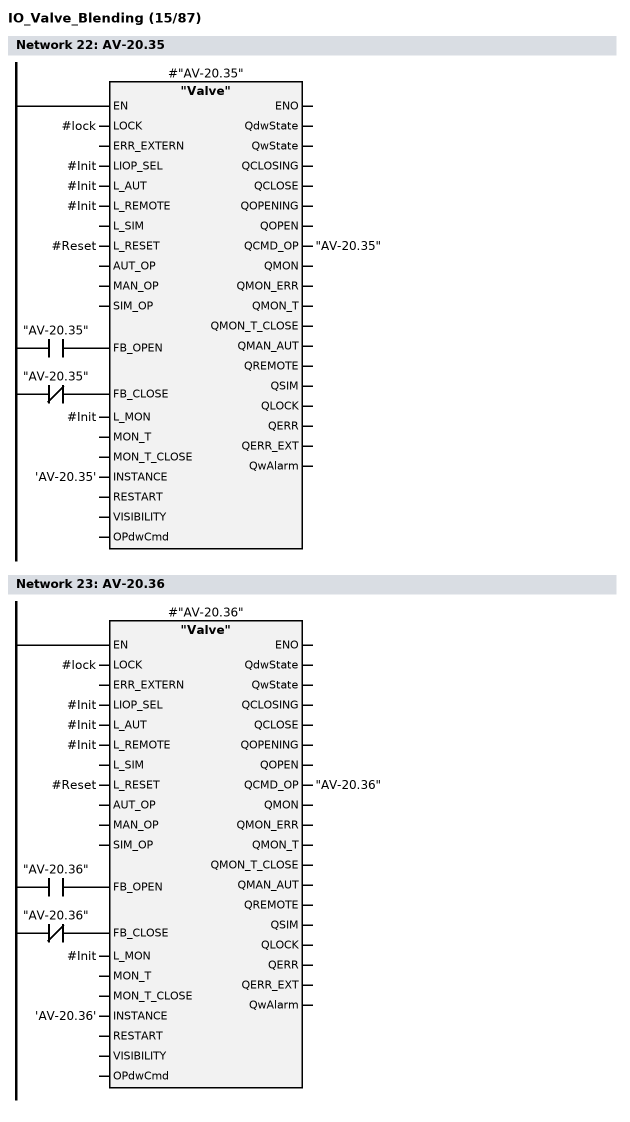
   RUNG wire#powerrail
      #"AV-20.35"(FB_OPEN := wire#w1, FB_CLOSE := wire#w2, LOCK := #lock, ERR_EXTERN :=, LIOP_SEL := #Init, L_AUT := #Init, L_REMOTE := #Init, L_SIM :=, L_RESET := #Reset, AUT_OP :=, MAN_OP :=, SIM_OP :=, L_MON := #Init, MON_T :=, MON_T_CLOSE :=, INSTANCE := 'AV-20.35', RESTART :=, VISIBILITY :=, OPdwCmd :=, QdwState =>, QwState =>, QCLOSING =>, QCLOSE =>, QOPENING =>, QOPEN =>, QCMD_OP => "AV-20.35", QMON =>, QMON_ERR =>, QMON_T =>, QMON_T_CLOSE =>, QMAN_AUT =>, QREMOTE =>, QSIM =>, QLOCK =>, QERR =>, QERR_EXT =>, QwAlarm =>)
   END_RUNG
   RUNG wire#powerrail
      Contact( "AV-20.35" )
   END_RUNG wire#w1
   RUNG wire#powerrail
      I_Contact( "AV-20.35" )
   END_RUNG wire#w2
   // the same network as SCL:
   #"AV-20.35"(LOCK := #lock,   // "Valve"
               LIOP_SEL := #Init,
               L_AUT := #Init,
               L_REMOTE := #Init,
               L_RESET := #Reset,
               FB_OPEN := "AV-20.35",
               FB_CLOSE := NOT "AV-20.35",
               L_MON := #Init,
               INSTANCE := 'AV-20.35',
               QCMD_OP => "AV-20.35");
END_REGION

REGION Network 23: AV-20.36
   RUNG wire#powerrail
      #"AV-20.36"(FB_OPEN := wire#w1, FB_CLOSE := wire#w2, LOCK := #lock, ERR_EXTERN :=, LIOP_SEL := #Init, L_AUT := #Init, L_REMOTE := #Init, L_SIM :=, L_RESET := #Reset, AUT_OP :=, MAN_OP :=, SIM_OP :=, L_MON := #Init, MON_T :=, MON_T_CLOSE :=, INSTANCE := 'AV-20.36', RESTART :=, VISIBILITY :=, OPdwCmd :=, QdwState =>, QwState =>, QCLOSING =>, QCLOSE =>, QOPENING =>, QOPEN =>, QCMD_OP => "AV-20.36", QMON =>, QMON_ERR =>, QMON_T =>, QMON_T_CLOSE =>, QMAN_AUT =>, QREMOTE =>, QSIM =>, QLOCK =>, QERR =>, QERR_EXT =>, QwAlarm =>)
   END_RUNG
   RUNG wire#powerrail
      Contact( "AV-20.36" )
   END_RUNG wire#w1
   RUNG wire#powerrail
      I_Contact( "AV-20.36" )
   END_RUNG wire#w2
   // the same network as SCL:
   #"AV-20.36"(LOCK := #lock,   // "Valve"
               LIOP_SEL := #Init,
               L_AUT := #Init,
               L_REMOTE := #Init,
               L_RESET := #Reset,
               FB_OPEN := "AV-20.36",
               FB_CLOSE := NOT "AV-20.36",
               L_MON := #Init,
               INSTANCE := 'AV-20.36',
               QCMD_OP => "AV-20.36");
END_REGION

REGION Network 24: AV-20.37
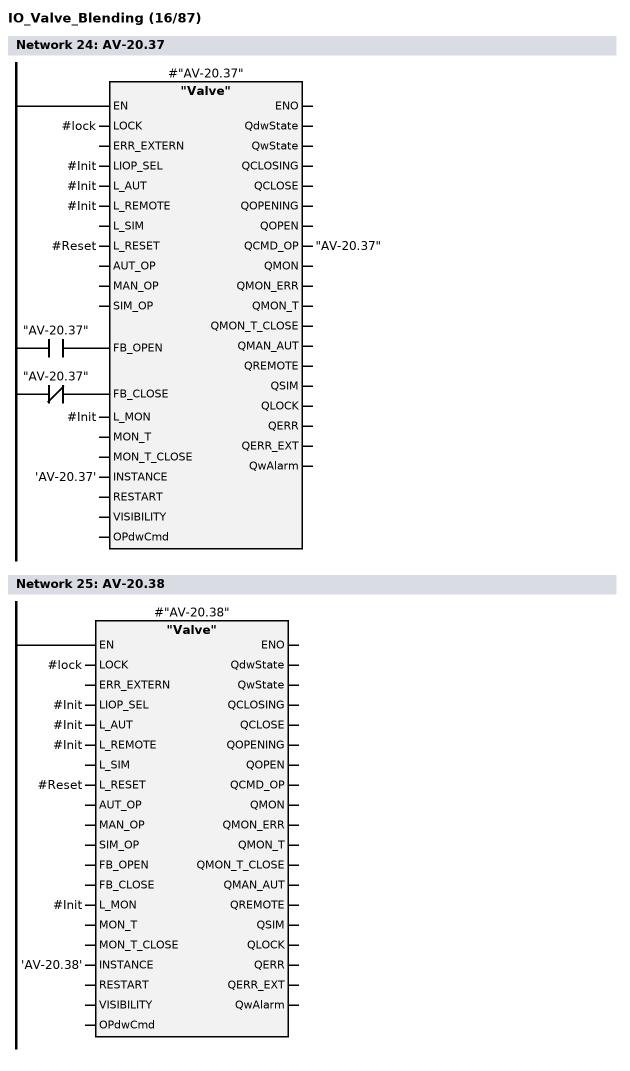
   RUNG wire#powerrail
      #"AV-20.37"(FB_OPEN := wire#w1, FB_CLOSE := wire#w2, LOCK := #lock, ERR_EXTERN :=, LIOP_SEL := #Init, L_AUT := #Init, L_REMOTE := #Init, L_SIM :=, L_RESET := #Reset, AUT_OP :=, MAN_OP :=, SIM_OP :=, L_MON := #Init, MON_T :=, MON_T_CLOSE :=, INSTANCE := 'AV-20.37', RESTART :=, VISIBILITY :=, OPdwCmd :=, QdwState =>, QwState =>, QCLOSING =>, QCLOSE =>, QOPENING =>, QOPEN =>, QCMD_OP => "AV-20.37", QMON =>, QMON_ERR =>, QMON_T =>, QMON_T_CLOSE =>, QMAN_AUT =>, QREMOTE =>, QSIM =>, QLOCK =>, QERR =>, QERR_EXT =>, QwAlarm =>)
   END_RUNG
   RUNG wire#powerrail
      Contact( "AV-20.37" )
   END_RUNG wire#w1
   RUNG wire#powerrail
      I_Contact( "AV-20.37" )
   END_RUNG wire#w2
   // the same network as SCL:
   #"AV-20.37"(LOCK := #lock,   // "Valve"
               LIOP_SEL := #Init,
               L_AUT := #Init,
               L_REMOTE := #Init,
               L_RESET := #Reset,
               FB_OPEN := "AV-20.37",
               FB_CLOSE := NOT "AV-20.37",
               L_MON := #Init,
               INSTANCE := 'AV-20.37',
               QCMD_OP => "AV-20.37");
END_REGION

REGION Network 25: AV-20.38
   RUNG wire#powerrail
      #"AV-20.38"(LOCK := #lock, ERR_EXTERN :=, LIOP_SEL := #Init, L_AUT := #Init, L_REMOTE := #Init, L_SIM :=, L_RESET := #Reset, AUT_OP :=, MAN_OP :=, SIM_OP :=, FB_OPEN :=, FB_CLOSE :=, L_MON := #Init, MON_T :=, MON_T_CLOSE :=, INSTANCE := 'AV-20.38', RESTART :=, VISIBILITY :=, OPdwCmd :=, QdwState =>, QwState =>, QCLOSING =>, QCLOSE =>, QOPENING =>, QOPEN =>, QCMD_OP =>, QMON =>, QMON_ERR =>, QMON_T =>, QMON_T_CLOSE =>, QMAN_AUT =>, QREMOTE =>, QSIM =>, QLOCK =>, QERR =>, QERR_EXT =>, QwAlarm =>)
   END_RUNG
   // the same network as SCL:
   #"AV-20.38"(LOCK := #lock,   // "Valve"
               LIOP_SEL := #Init,
               L_AUT := #Init,
               L_REMOTE := #Init,
               L_RESET := #Reset,
               L_MON := #Init,
               INSTANCE := 'AV-20.38');
END_REGION

REGION Network 26: AV-20.39
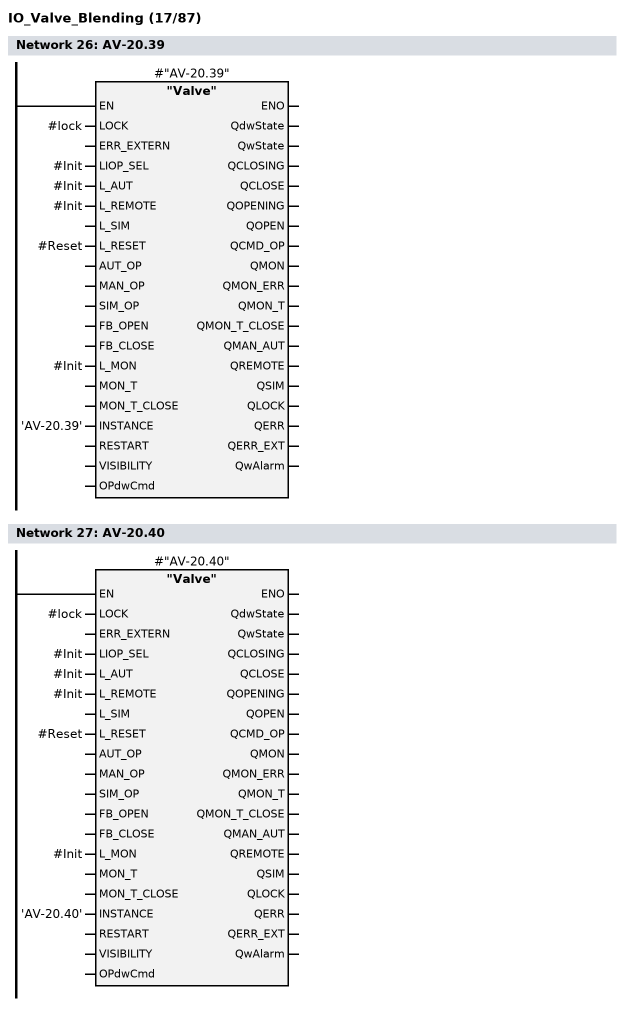
   RUNG wire#powerrail
      #"AV-20.39"(LOCK := #lock, ERR_EXTERN :=, LIOP_SEL := #Init, L_AUT := #Init, L_REMOTE := #Init, L_SIM :=, L_RESET := #Reset, AUT_OP :=, MAN_OP :=, SIM_OP :=, FB_OPEN :=, FB_CLOSE :=, L_MON := #Init, MON_T :=, MON_T_CLOSE :=, INSTANCE := 'AV-20.39', RESTART :=, VISIBILITY :=, OPdwCmd :=, QdwState =>, QwState =>, QCLOSING =>, QCLOSE =>, QOPENING =>, QOPEN =>, QCMD_OP =>, QMON =>, QMON_ERR =>, QMON_T =>, QMON_T_CLOSE =>, QMAN_AUT =>, QREMOTE =>, QSIM =>, QLOCK =>, QERR =>, QERR_EXT =>, QwAlarm =>)
   END_RUNG
   // the same network as SCL:
   #"AV-20.39"(LOCK := #lock,   // "Valve"
               LIOP_SEL := #Init,
               L_AUT := #Init,
               L_REMOTE := #Init,
               L_RESET := #Reset,
               L_MON := #Init,
               INSTANCE := 'AV-20.39');
END_REGION

REGION Network 27: AV-20.40
   RUNG wire#powerrail
      #"AV-20.40"(LOCK := #lock, ERR_EXTERN :=, LIOP_SEL := #Init, L_AUT := #Init, L_REMOTE := #Init, L_SIM :=, L_RESET := #Reset, AUT_OP :=, MAN_OP :=, SIM_OP :=, FB_OPEN :=, FB_CLOSE :=, L_MON := #Init, MON_T :=, MON_T_CLOSE :=, INSTANCE := 'AV-20.40', RESTART :=, VISIBILITY :=, OPdwCmd :=, QdwState =>, QwState =>, QCLOSING =>, QCLOSE =>, QOPENING =>, QOPEN =>, QCMD_OP =>, QMON =>, QMON_ERR =>, QMON_T =>, QMON_T_CLOSE =>, QMAN_AUT =>, QREMOTE =>, QSIM =>, QLOCK =>, QERR =>, QERR_EXT =>, QwAlarm =>)
   END_RUNG
   // the same network as SCL:
   #"AV-20.40"(LOCK := #lock,   // "Valve"
               LIOP_SEL := #Init,
               L_AUT := #Init,
               L_REMOTE := #Init,
               L_RESET := #Reset,
               L_MON := #Init,
               INSTANCE := 'AV-20.40');
END_REGION

REGION Network 28: AV-20.41
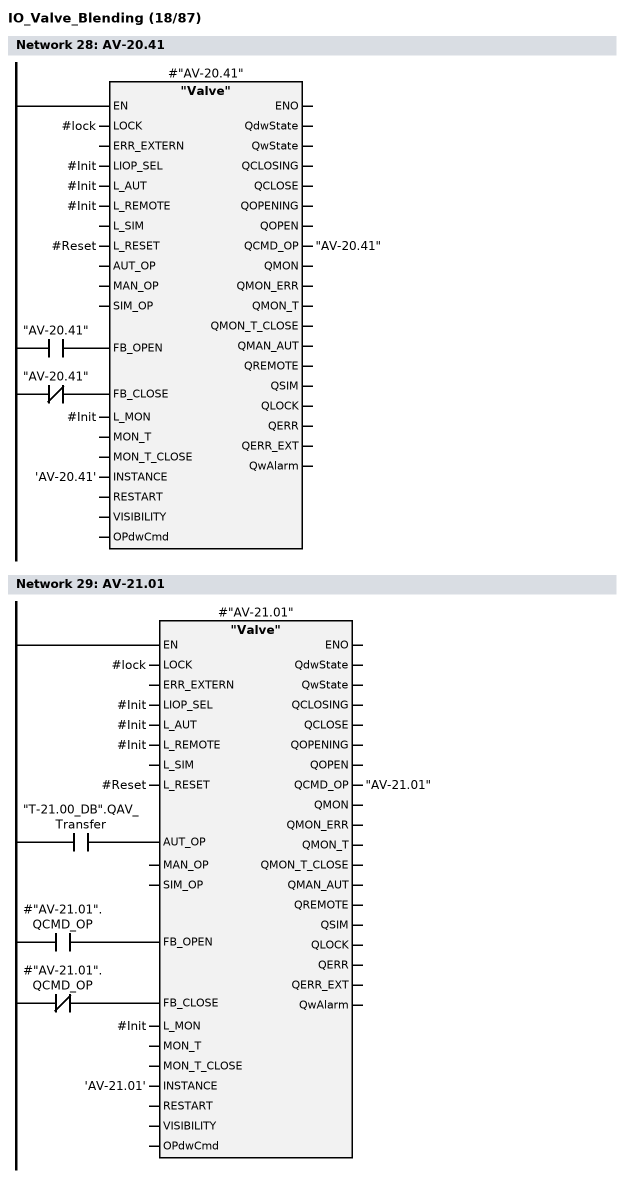
   RUNG wire#powerrail
      #"AV-20.41"(FB_OPEN := wire#w1, FB_CLOSE := wire#w2, LOCK := #lock, ERR_EXTERN :=, LIOP_SEL := #Init, L_AUT := #Init, L_REMOTE := #Init, L_SIM :=, L_RESET := #Reset, AUT_OP :=, MAN_OP :=, SIM_OP :=, L_MON := #Init, MON_T :=, MON_T_CLOSE :=, INSTANCE := 'AV-20.41', RESTART :=, VISIBILITY :=, OPdwCmd :=, QdwState =>, QwState =>, QCLOSING =>, QCLOSE =>, QOPENING =>, QOPEN =>, QCMD_OP => "AV-20.41", QMON =>, QMON_ERR =>, QMON_T =>, QMON_T_CLOSE =>, QMAN_AUT =>, QREMOTE =>, QSIM =>, QLOCK =>, QERR =>, QERR_EXT =>, QwAlarm =>)
   END_RUNG
   RUNG wire#powerrail
      Contact( "AV-20.41" )
   END_RUNG wire#w1
   RUNG wire#powerrail
      I_Contact( "AV-20.41" )
   END_RUNG wire#w2
   // the same network as SCL:
   #"AV-20.41"(LOCK := #lock,   // "Valve"
               LIOP_SEL := #Init,
               L_AUT := #Init,
               L_REMOTE := #Init,
               L_RESET := #Reset,
               FB_OPEN := "AV-20.41",
               FB_CLOSE := NOT "AV-20.41",
               L_MON := #Init,
               INSTANCE := 'AV-20.41',
               QCMD_OP => "AV-20.41");
END_REGION

REGION Network 29: AV-21.01
   RUNG wire#powerrail
      #"AV-21.01"(AUT_OP := wire#w1, FB_OPEN := wire#w2, FB_CLOSE := wire#w3, LOCK := #lock, ERR_EXTERN :=, LIOP_SEL := #Init, L_AUT := #Init, L_REMOTE := #Init, L_SIM :=, L_RESET := #Reset, MAN_OP :=, SIM_OP :=, L_MON := #Init, MON_T :=, MON_T_CLOSE :=, INSTANCE := 'AV-21.01', RESTART :=, VISIBILITY :=, OPdwCmd :=, QdwState =>, QwState =>, QCLOSING =>, QCLOSE =>, QOPENING =>, QOPEN =>, QCMD_OP => "AV-21.01", QMON =>, QMON_ERR =>, QMON_T =>, QMON_T_CLOSE =>, QMAN_AUT =>, QREMOTE =>, QSIM =>, QLOCK =>, QERR =>, QERR_EXT =>, QwAlarm =>)
   END_RUNG
   RUNG wire#powerrail
      Contact( "T-21.00_DB".QAV_Transfer )
   END_RUNG wire#w1
   RUNG wire#powerrail
      Contact( #"AV-21.01".QCMD_OP )
   END_RUNG wire#w2
   RUNG wire#powerrail
      I_Contact( #"AV-21.01".QCMD_OP )
   END_RUNG wire#w3
   // the same network as SCL:
   #"AV-21.01"(LOCK := #lock,   // "Valve"
               LIOP_SEL := #Init,
               L_AUT := #Init,
               L_REMOTE := #Init,
               L_RESET := #Reset,
               AUT_OP := "T-21.00_DB".QAV_Transfer,
               FB_OPEN := #"AV-21.01".QCMD_OP,
               FB_CLOSE := NOT #"AV-21.01".QCMD_OP,
               L_MON := #Init,
               INSTANCE := 'AV-21.01',
               QCMD_OP => "AV-21.01");
END_REGION

REGION Network 30: AV-21.02
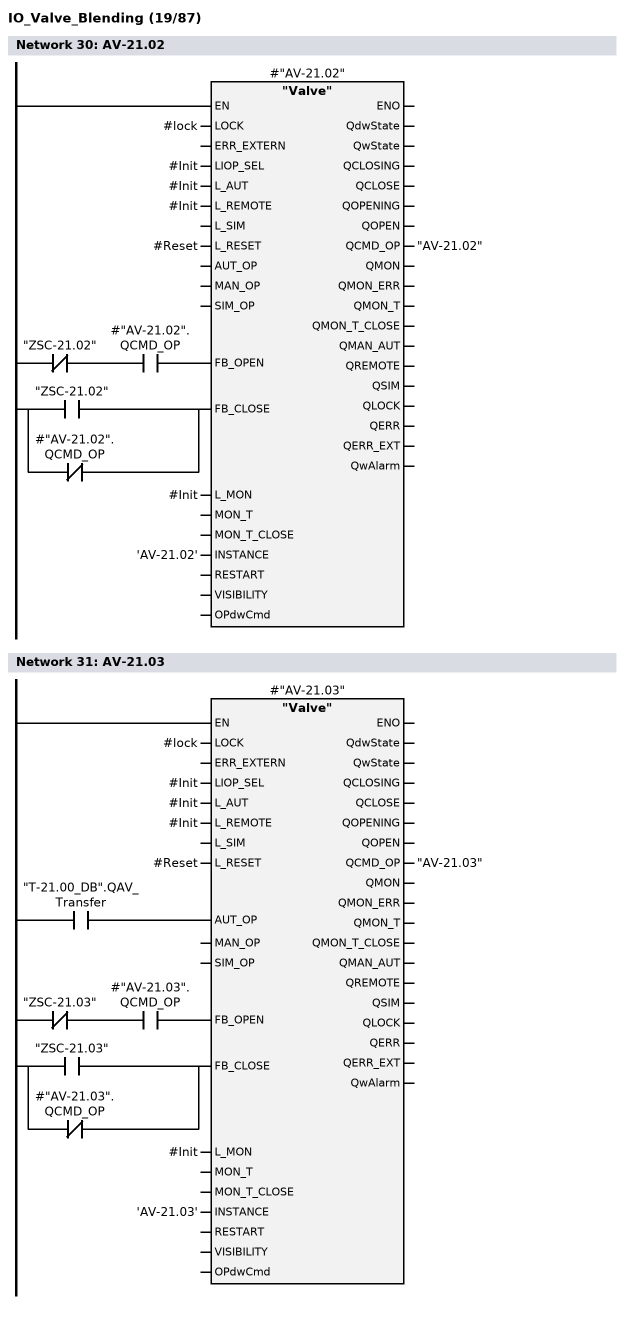
   RUNG wire#powerrail
      #"AV-21.02"(FB_OPEN := wire#w1, FB_CLOSE := wire#w2, LOCK := #lock, ERR_EXTERN :=, LIOP_SEL := #Init, L_AUT := #Init, L_REMOTE := #Init, L_SIM :=, L_RESET := #Reset, AUT_OP :=, MAN_OP :=, SIM_OP :=, L_MON := #Init, MON_T :=, MON_T_CLOSE :=, INSTANCE := 'AV-21.02', RESTART :=, VISIBILITY :=, OPdwCmd :=, QdwState =>, QwState =>, QCLOSING =>, QCLOSE =>, QOPENING =>, QOPEN =>, QCMD_OP => "AV-21.02", QMON =>, QMON_ERR =>, QMON_T =>, QMON_T_CLOSE =>, QMAN_AUT =>, QREMOTE =>, QSIM =>, QLOCK =>, QERR =>, QERR_EXT =>, QwAlarm =>)
   END_RUNG
   RUNG wire#powerrail
      I_Contact( "ZSC-21.02" )
      Contact( #"AV-21.02".QCMD_OP )
   END_RUNG wire#w1
   RUNG wire#powerrail
      Contact( "ZSC-21.02" )
   END_RUNG wire#w2
   RUNG wire#powerrail
      I_Contact( #"AV-21.02".QCMD_OP )
   END_RUNG wire#w2
   // the same network as SCL:
   #"AV-21.02"(LOCK := #lock,   // "Valve"
               LIOP_SEL := #Init,
               L_AUT := #Init,
               L_REMOTE := #Init,
               L_RESET := #Reset,
               FB_OPEN := NOT "ZSC-21.02" AND #"AV-21.02".QCMD_OP,
               FB_CLOSE := "ZSC-21.02" OR NOT #"AV-21.02".QCMD_OP,
               L_MON := #Init,
               INSTANCE := 'AV-21.02',
               QCMD_OP => "AV-21.02");
END_REGION

REGION Network 31: AV-21.03
   RUNG wire#powerrail
      #"AV-21.03"(AUT_OP := wire#w1, FB_OPEN := wire#w2, FB_CLOSE := wire#w3, LOCK := #lock, ERR_EXTERN :=, LIOP_SEL := #Init, L_AUT := #Init, L_REMOTE := #Init, L_SIM :=, L_RESET := #Reset, MAN_OP :=, SIM_OP :=, L_MON := #Init, MON_T :=, MON_T_CLOSE :=, INSTANCE := 'AV-21.03', RESTART :=, VISIBILITY :=, OPdwCmd :=, QdwState =>, QwState =>, QCLOSING =>, QCLOSE =>, QOPENING =>, QOPEN =>, QCMD_OP => "AV-21.03", QMON =>, QMON_ERR =>, QMON_T =>, QMON_T_CLOSE =>, QMAN_AUT =>, QREMOTE =>, QSIM =>, QLOCK =>, QERR =>, QERR_EXT =>, QwAlarm =>)
   END_RUNG
   RUNG wire#powerrail
      Contact( "T-21.00_DB".QAV_Transfer )
   END_RUNG wire#w1
   RUNG wire#powerrail
      I_Contact( "ZSC-21.03" )
      Contact( #"AV-21.03".QCMD_OP )
   END_RUNG wire#w2
   RUNG wire#powerrail
      Contact( "ZSC-21.03" )
   END_RUNG wire#w3
   RUNG wire#powerrail
      I_Contact( #"AV-21.03".QCMD_OP )
   END_RUNG wire#w3
   // the same network as SCL:
   #"AV-21.03"(LOCK := #lock,   // "Valve"
               LIOP_SEL := #Init,
               L_AUT := #Init,
               L_REMOTE := #Init,
               L_RESET := #Reset,
               AUT_OP := "T-21.00_DB".QAV_Transfer,
               FB_OPEN := NOT "ZSC-21.03" AND #"AV-21.03".QCMD_OP,
               FB_CLOSE := "ZSC-21.03" OR NOT #"AV-21.03".QCMD_OP,
               L_MON := #Init,
               INSTANCE := 'AV-21.03',
               QCMD_OP => "AV-21.03");
END_REGION

REGION Network 32: AV-21.04
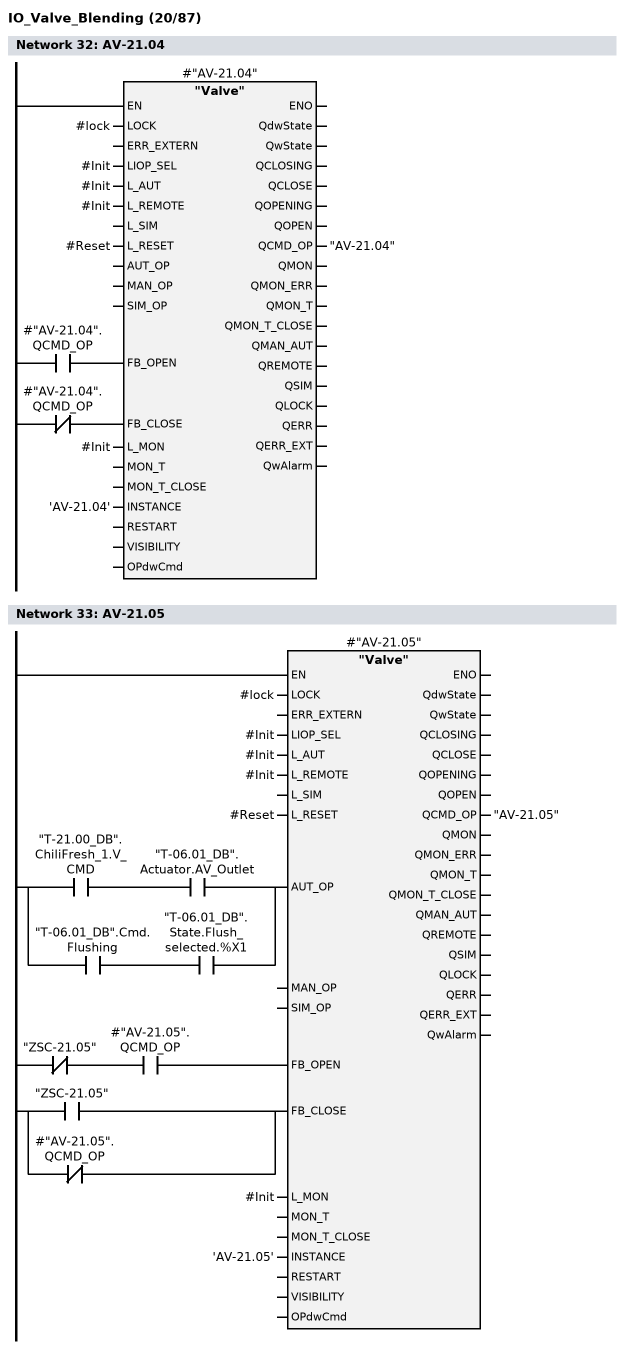
   RUNG wire#powerrail
      #"AV-21.04"(FB_OPEN := wire#w1, FB_CLOSE := wire#w2, LOCK := #lock, ERR_EXTERN :=, LIOP_SEL := #Init, L_AUT := #Init, L_REMOTE := #Init, L_SIM :=, L_RESET := #Reset, AUT_OP :=, MAN_OP :=, SIM_OP :=, L_MON := #Init, MON_T :=, MON_T_CLOSE :=, INSTANCE := 'AV-21.04', RESTART :=, VISIBILITY :=, OPdwCmd :=, QdwState =>, QwState =>, QCLOSING =>, QCLOSE =>, QOPENING =>, QOPEN =>, QCMD_OP => "AV-21.04", QMON =>, QMON_ERR =>, QMON_T =>, QMON_T_CLOSE =>, QMAN_AUT =>, QREMOTE =>, QSIM =>, QLOCK =>, QERR =>, QERR_EXT =>, QwAlarm =>)
   END_RUNG
   RUNG wire#powerrail
      Contact( #"AV-21.04".QCMD_OP )
   END_RUNG wire#w1
   RUNG wire#powerrail
      I_Contact( #"AV-21.04".QCMD_OP )
   END_RUNG wire#w2
   // the same network as SCL:
   #"AV-21.04"(LOCK := #lock,   // "Valve"
               LIOP_SEL := #Init,
               L_AUT := #Init,
               L_REMOTE := #Init,
               L_RESET := #Reset,
               FB_OPEN := #"AV-21.04".QCMD_OP,
               FB_CLOSE := NOT #"AV-21.04".QCMD_OP,
               L_MON := #Init,
               INSTANCE := 'AV-21.04',
               QCMD_OP => "AV-21.04");
END_REGION

REGION Network 33: AV-21.05
   RUNG wire#powerrail
      #"AV-21.05"(AUT_OP := wire#w1, FB_OPEN := wire#w2, FB_CLOSE := wire#w3, LOCK := #lock, ERR_EXTERN :=, LIOP_SEL := #Init, L_AUT := #Init, L_REMOTE := #Init, L_SIM :=, L_RESET := #Reset, MAN_OP :=, SIM_OP :=, L_MON := #Init, MON_T :=, MON_T_CLOSE :=, INSTANCE := 'AV-21.05', RESTART :=, VISIBILITY :=, OPdwCmd :=, QdwState =>, QwState =>, QCLOSING =>, QCLOSE =>, QOPENING =>, QOPEN =>, QCMD_OP => "AV-21.05", QMON =>, QMON_ERR =>, QMON_T =>, QMON_T_CLOSE =>, QMAN_AUT =>, QREMOTE =>, QSIM =>, QLOCK =>, QERR =>, QERR_EXT =>, QwAlarm =>)
   END_RUNG
   RUNG wire#powerrail
      Contact( "T-21.00_DB".ChiliFresh_1.V_CMD )
      Contact( "T-06.01_DB".Actuator.AV_Outlet )
   END_RUNG wire#w1
   RUNG wire#powerrail
      Contact( "T-06.01_DB".Cmd.Flushing )
      Contact( "T-06.01_DB".State.Flush_selected.%X1 )
   END_RUNG wire#w1
   RUNG wire#powerrail
      I_Contact( "ZSC-21.05" )
      Contact( #"AV-21.05".QCMD_OP )
   END_RUNG wire#w2
   RUNG wire#powerrail
      Contact( "ZSC-21.05" )
   END_RUNG wire#w3
   RUNG wire#powerrail
      I_Contact( #"AV-21.05".QCMD_OP )
   END_RUNG wire#w3
   // the same network as SCL:
   #"AV-21.05"(LOCK := #lock,   // "Valve"
               LIOP_SEL := #Init,
               L_AUT := #Init,
               L_REMOTE := #Init,
               L_RESET := #Reset,
               AUT_OP := ("T-21.00_DB".ChiliFresh_1.V_CMD AND "T-06.01_DB".Actuator.AV_Outlet) OR ("T-06.01_DB".Cmd.Flushing AND "T-06.01_DB".State.Flush_selected.%X1),
               FB_OPEN := NOT "ZSC-21.05" AND #"AV-21.05".QCMD_OP,
               FB_CLOSE := "ZSC-21.05" OR NOT #"AV-21.05".QCMD_OP,
               L_MON := #Init,
               INSTANCE := 'AV-21.05',
               QCMD_OP => "AV-21.05");
END_REGION

REGION Network 34: AV-21.06
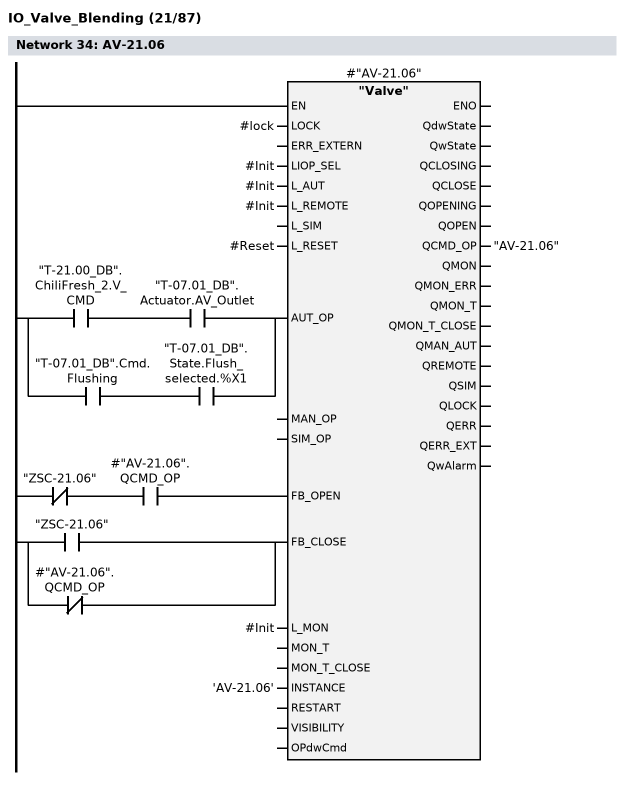
   RUNG wire#powerrail
      #"AV-21.06"(AUT_OP := wire#w1, FB_OPEN := wire#w2, FB_CLOSE := wire#w3, LOCK := #lock, ERR_EXTERN :=, LIOP_SEL := #Init, L_AUT := #Init, L_REMOTE := #Init, L_SIM :=, L_RESET := #Reset, MAN_OP :=, SIM_OP :=, L_MON := #Init, MON_T :=, MON_T_CLOSE :=, INSTANCE := 'AV-21.06', RESTART :=, VISIBILITY :=, OPdwCmd :=, QdwState =>, QwState =>, QCLOSING =>, QCLOSE =>, QOPENING =>, QOPEN =>, QCMD_OP => "AV-21.06", QMON =>, QMON_ERR =>, QMON_T =>, QMON_T_CLOSE =>, QMAN_AUT =>, QREMOTE =>, QSIM =>, QLOCK =>, QERR =>, QERR_EXT =>, QwAlarm =>)
   END_RUNG
   RUNG wire#powerrail
      Contact( "T-21.00_DB".ChiliFresh_2.V_CMD )
      Contact( "T-07.01_DB".Actuator.AV_Outlet )
   END_RUNG wire#w1
   RUNG wire#powerrail
      Contact( "T-07.01_DB".Cmd.Flushing )
      Contact( "T-07.01_DB".State.Flush_selected.%X1 )
   END_RUNG wire#w1
   RUNG wire#powerrail
      I_Contact( "ZSC-21.06" )
      Contact( #"AV-21.06".QCMD_OP )
   END_RUNG wire#w2
   RUNG wire#powerrail
      Contact( "ZSC-21.06" )
   END_RUNG wire#w3
   RUNG wire#powerrail
      I_Contact( #"AV-21.06".QCMD_OP )
   END_RUNG wire#w3
   // the same network as SCL:
   #"AV-21.06"(LOCK := #lock,   // "Valve"
               LIOP_SEL := #Init,
               L_AUT := #Init,
               L_REMOTE := #Init,
               L_RESET := #Reset,
               AUT_OP := ("T-21.00_DB".ChiliFresh_2.V_CMD AND "T-07.01_DB".Actuator.AV_Outlet) OR ("T-07.01_DB".Cmd.Flushing AND "T-07.01_DB".State.Flush_selected.%X1),
               FB_OPEN := NOT "ZSC-21.06" AND #"AV-21.06".QCMD_OP,
               FB_CLOSE := "ZSC-21.06" OR NOT #"AV-21.06".QCMD_OP,
               L_MON := #Init,
               INSTANCE := 'AV-21.06',
               QCMD_OP => "AV-21.06");
END_REGION

REGION Network 35: AV-21.07
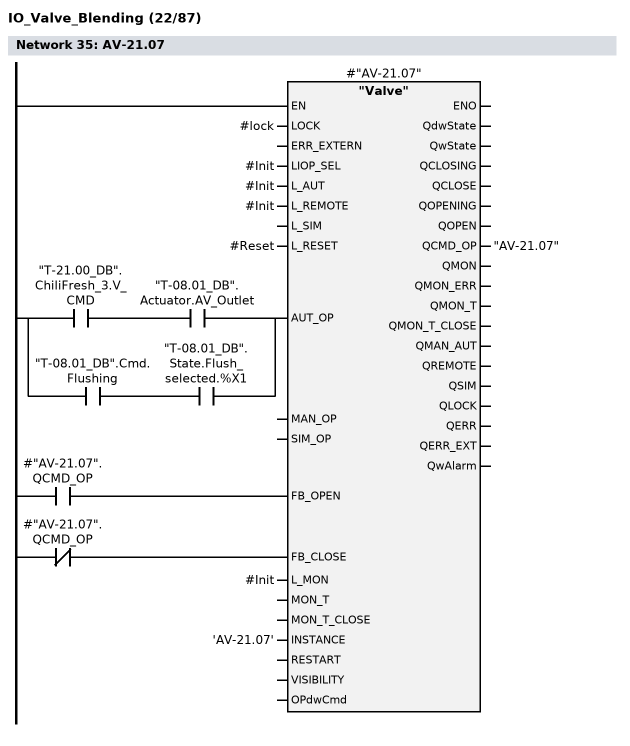
   RUNG wire#powerrail
      #"AV-21.07"(AUT_OP := wire#w1, FB_OPEN := wire#w2, FB_CLOSE := wire#w3, LOCK := #lock, ERR_EXTERN :=, LIOP_SEL := #Init, L_AUT := #Init, L_REMOTE := #Init, L_SIM :=, L_RESET := #Reset, MAN_OP :=, SIM_OP :=, L_MON := #Init, MON_T :=, MON_T_CLOSE :=, INSTANCE := 'AV-21.07', RESTART :=, VISIBILITY :=, OPdwCmd :=, QdwState =>, QwState =>, QCLOSING =>, QCLOSE =>, QOPENING =>, QOPEN =>, QCMD_OP => "AV-21.07", QMON =>, QMON_ERR =>, QMON_T =>, QMON_T_CLOSE =>, QMAN_AUT =>, QREMOTE =>, QSIM =>, QLOCK =>, QERR =>, QERR_EXT =>, QwAlarm =>)
   END_RUNG
   RUNG wire#powerrail
      Contact( "T-21.00_DB".ChiliFresh_3.V_CMD )
      Contact( "T-08.01_DB".Actuator.AV_Outlet )
   END_RUNG wire#w1
   RUNG wire#powerrail
      Contact( "T-08.01_DB".Cmd.Flushing )
      Contact( "T-08.01_DB".State.Flush_selected.%X1 )
   END_RUNG wire#w1
   RUNG wire#powerrail
      Contact( #"AV-21.07".QCMD_OP )
   END_RUNG wire#w2
   RUNG wire#powerrail
      I_Contact( #"AV-21.07".QCMD_OP )
   END_RUNG wire#w3
   // the same network as SCL:
   #"AV-21.07"(LOCK := #lock,   // "Valve"
               LIOP_SEL := #Init,
               L_AUT := #Init,
               L_REMOTE := #Init,
               L_RESET := #Reset,
               AUT_OP := ("T-21.00_DB".ChiliFresh_3.V_CMD AND "T-08.01_DB".Actuator.AV_Outlet) OR ("T-08.01_DB".Cmd.Flushing AND "T-08.01_DB".State.Flush_selected.%X1),
               FB_OPEN := #"AV-21.07".QCMD_OP,
               FB_CLOSE := NOT #"AV-21.07".QCMD_OP,
               L_MON := #Init,
               INSTANCE := 'AV-21.07',
               QCMD_OP => "AV-21.07");
END_REGION

REGION Network 36: AV-21.08
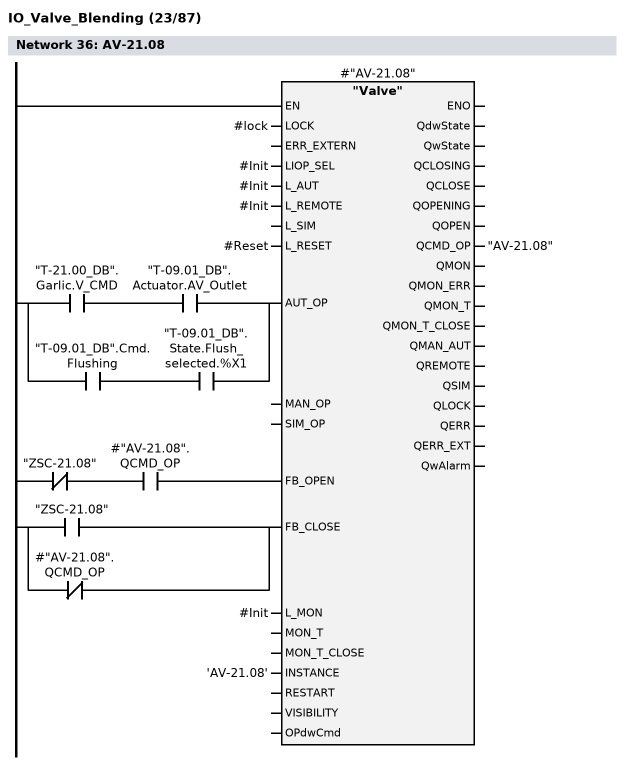
   RUNG wire#powerrail
      #"AV-21.08"(AUT_OP := wire#w1, FB_OPEN := wire#w2, FB_CLOSE := wire#w3, LOCK := #lock, ERR_EXTERN :=, LIOP_SEL := #Init, L_AUT := #Init, L_REMOTE := #Init, L_SIM :=, L_RESET := #Reset, MAN_OP :=, SIM_OP :=, L_MON := #Init, MON_T :=, MON_T_CLOSE :=, INSTANCE := 'AV-21.08', RESTART :=, VISIBILITY :=, OPdwCmd :=, QdwState =>, QwState =>, QCLOSING =>, QCLOSE =>, QOPENING =>, QOPEN =>, QCMD_OP => "AV-21.08", QMON =>, QMON_ERR =>, QMON_T =>, QMON_T_CLOSE =>, QMAN_AUT =>, QREMOTE =>, QSIM =>, QLOCK =>, QERR =>, QERR_EXT =>, QwAlarm =>)
   END_RUNG
   RUNG wire#powerrail
      Contact( "T-21.00_DB".Garlic.V_CMD )
      Contact( "T-09.01_DB".Actuator.AV_Outlet )
   END_RUNG wire#w1
   RUNG wire#powerrail
      Contact( "T-09.01_DB".Cmd.Flushing )
      Contact( "T-09.01_DB".State.Flush_selected.%X1 )
   END_RUNG wire#w1
   RUNG wire#powerrail
      I_Contact( "ZSC-21.08" )
      Contact( #"AV-21.08".QCMD_OP )
   END_RUNG wire#w2
   RUNG wire#powerrail
      Contact( "ZSC-21.08" )
   END_RUNG wire#w3
   RUNG wire#powerrail
      I_Contact( #"AV-21.08".QCMD_OP )
   END_RUNG wire#w3
   // the same network as SCL:
   #"AV-21.08"(LOCK := #lock,   // "Valve"
               LIOP_SEL := #Init,
               L_AUT := #Init,
               L_REMOTE := #Init,
               L_RESET := #Reset,
               AUT_OP := ("T-21.00_DB".Garlic.V_CMD AND "T-09.01_DB".Actuator.AV_Outlet) OR ("T-09.01_DB".Cmd.Flushing AND "T-09.01_DB".State.Flush_selected.%X1),
               FB_OPEN := NOT "ZSC-21.08" AND #"AV-21.08".QCMD_OP,
               FB_CLOSE := "ZSC-21.08" OR NOT #"AV-21.08".QCMD_OP,
               L_MON := #Init,
               INSTANCE := 'AV-21.08',
               QCMD_OP => "AV-21.08");
END_REGION

REGION Network 37: AV-21.09
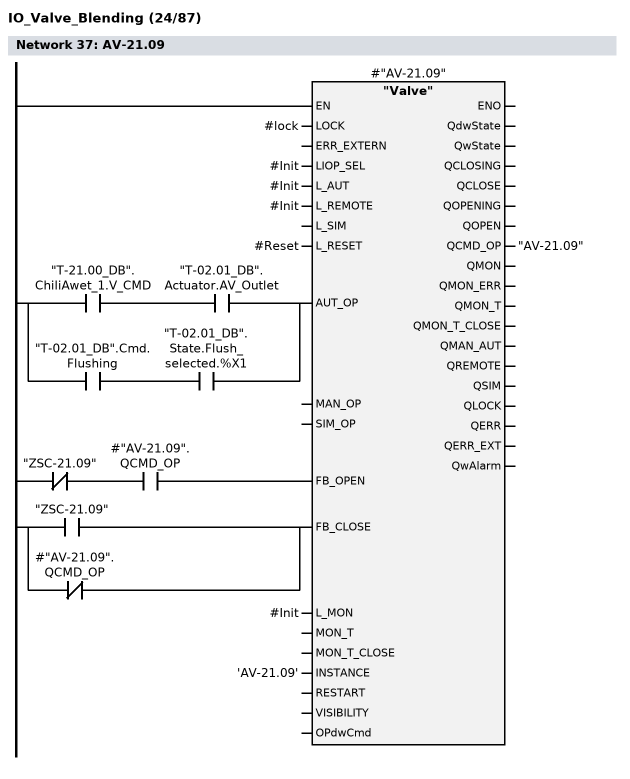
   RUNG wire#powerrail
      #"AV-21.09"(AUT_OP := wire#w1, FB_OPEN := wire#w2, FB_CLOSE := wire#w3, LOCK := #lock, ERR_EXTERN :=, LIOP_SEL := #Init, L_AUT := #Init, L_REMOTE := #Init, L_SIM :=, L_RESET := #Reset, MAN_OP :=, SIM_OP :=, L_MON := #Init, MON_T :=, MON_T_CLOSE :=, INSTANCE := 'AV-21.09', RESTART :=, VISIBILITY :=, OPdwCmd :=, QdwState =>, QwState =>, QCLOSING =>, QCLOSE =>, QOPENING =>, QOPEN =>, QCMD_OP => "AV-21.09", QMON =>, QMON_ERR =>, QMON_T =>, QMON_T_CLOSE =>, QMAN_AUT =>, QREMOTE =>, QSIM =>, QLOCK =>, QERR =>, QERR_EXT =>, QwAlarm =>)
   END_RUNG
   RUNG wire#powerrail
      Contact( "T-21.00_DB".ChiliAwet_1.V_CMD )
      Contact( "T-02.01_DB".Actuator.AV_Outlet )
   END_RUNG wire#w1
   RUNG wire#powerrail
      Contact( "T-02.01_DB".Cmd.Flushing )
      Contact( "T-02.01_DB".State.Flush_selected.%X1 )
   END_RUNG wire#w1
   RUNG wire#powerrail
      I_Contact( "ZSC-21.09" )
      Contact( #"AV-21.09".QCMD_OP )
   END_RUNG wire#w2
   RUNG wire#powerrail
      Contact( "ZSC-21.09" )
   END_RUNG wire#w3
   RUNG wire#powerrail
      I_Contact( #"AV-21.09".QCMD_OP )
   END_RUNG wire#w3
   // the same network as SCL:
   #"AV-21.09"(LOCK := #lock,   // "Valve"
               LIOP_SEL := #Init,
               L_AUT := #Init,
               L_REMOTE := #Init,
               L_RESET := #Reset,
               AUT_OP := ("T-21.00_DB".ChiliAwet_1.V_CMD AND "T-02.01_DB".Actuator.AV_Outlet) OR ("T-02.01_DB".Cmd.Flushing AND "T-02.01_DB".State.Flush_selected.%X1),
               FB_OPEN := NOT "ZSC-21.09" AND #"AV-21.09".QCMD_OP,
               FB_CLOSE := "ZSC-21.09" OR NOT #"AV-21.09".QCMD_OP,
               L_MON := #Init,
               INSTANCE := 'AV-21.09',
               QCMD_OP => "AV-21.09");
END_REGION

REGION Network 38: AV-21.10
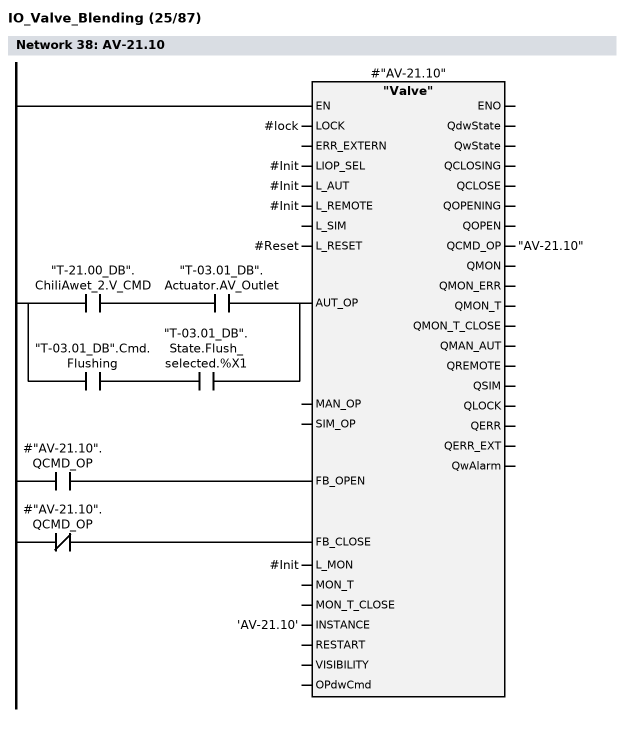
   RUNG wire#powerrail
      #"AV-21.10"(AUT_OP := wire#w1, FB_OPEN := wire#w2, FB_CLOSE := wire#w3, LOCK := #lock, ERR_EXTERN :=, LIOP_SEL := #Init, L_AUT := #Init, L_REMOTE := #Init, L_SIM :=, L_RESET := #Reset, MAN_OP :=, SIM_OP :=, L_MON := #Init, MON_T :=, MON_T_CLOSE :=, INSTANCE := 'AV-21.10', RESTART :=, VISIBILITY :=, OPdwCmd :=, QdwState =>, QwState =>, QCLOSING =>, QCLOSE =>, QOPENING =>, QOPEN =>, QCMD_OP => "AV-21.10", QMON =>, QMON_ERR =>, QMON_T =>, QMON_T_CLOSE =>, QMAN_AUT =>, QREMOTE =>, QSIM =>, QLOCK =>, QERR =>, QERR_EXT =>, QwAlarm =>)
   END_RUNG
   RUNG wire#powerrail
      Contact( "T-21.00_DB".ChiliAwet_2.V_CMD )
      Contact( "T-03.01_DB".Actuator.AV_Outlet )
   END_RUNG wire#w1
   RUNG wire#powerrail
      Contact( "T-03.01_DB".Cmd.Flushing )
      Contact( "T-03.01_DB".State.Flush_selected.%X1 )
   END_RUNG wire#w1
   RUNG wire#powerrail
      Contact( #"AV-21.10".QCMD_OP )
   END_RUNG wire#w2
   RUNG wire#powerrail
      I_Contact( #"AV-21.10".QCMD_OP )
   END_RUNG wire#w3
   // the same network as SCL:
   #"AV-21.10"(LOCK := #lock,   // "Valve"
               LIOP_SEL := #Init,
               L_AUT := #Init,
               L_REMOTE := #Init,
               L_RESET := #Reset,
               AUT_OP := ("T-21.00_DB".ChiliAwet_2.V_CMD AND "T-03.01_DB".Actuator.AV_Outlet) OR ("T-03.01_DB".Cmd.Flushing AND "T-03.01_DB".State.Flush_selected.%X1),
               FB_OPEN := #"AV-21.10".QCMD_OP,
               FB_CLOSE := NOT #"AV-21.10".QCMD_OP,
               L_MON := #Init,
               INSTANCE := 'AV-21.10',
               QCMD_OP => "AV-21.10");
END_REGION

REGION Network 39: AV-21.11
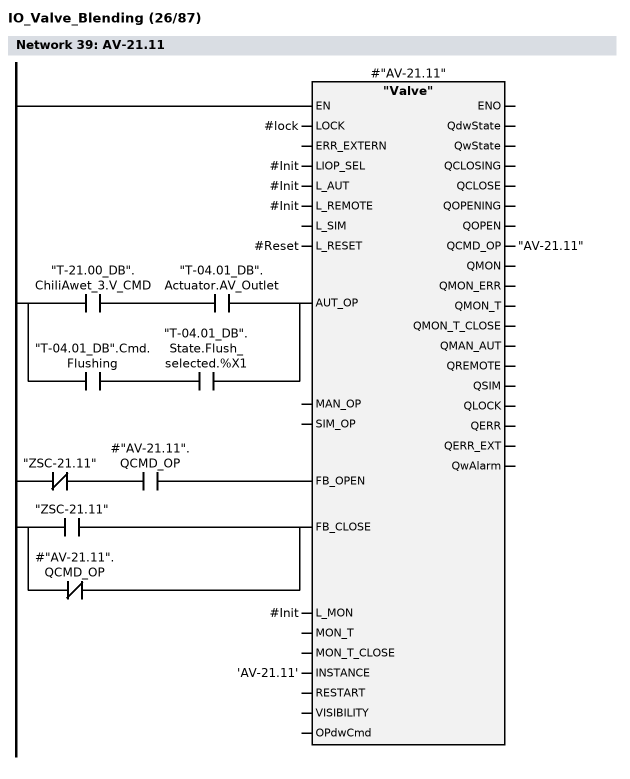
   RUNG wire#powerrail
      #"AV-21.11"(AUT_OP := wire#w1, FB_OPEN := wire#w2, FB_CLOSE := wire#w3, LOCK := #lock, ERR_EXTERN :=, LIOP_SEL := #Init, L_AUT := #Init, L_REMOTE := #Init, L_SIM :=, L_RESET := #Reset, MAN_OP :=, SIM_OP :=, L_MON := #Init, MON_T :=, MON_T_CLOSE :=, INSTANCE := 'AV-21.11', RESTART :=, VISIBILITY :=, OPdwCmd :=, QdwState =>, QwState =>, QCLOSING =>, QCLOSE =>, QOPENING =>, QOPEN =>, QCMD_OP => "AV-21.11", QMON =>, QMON_ERR =>, QMON_T =>, QMON_T_CLOSE =>, QMAN_AUT =>, QREMOTE =>, QSIM =>, QLOCK =>, QERR =>, QERR_EXT =>, QwAlarm =>)
   END_RUNG
   RUNG wire#powerrail
      Contact( "T-21.00_DB".ChiliAwet_3.V_CMD )
      Contact( "T-04.01_DB".Actuator.AV_Outlet )
   END_RUNG wire#w1
   RUNG wire#powerrail
      Contact( "T-04.01_DB".Cmd.Flushing )
      Contact( "T-04.01_DB".State.Flush_selected.%X1 )
   END_RUNG wire#w1
   RUNG wire#powerrail
      I_Contact( "ZSC-21.11" )
      Contact( #"AV-21.11".QCMD_OP )
   END_RUNG wire#w2
   RUNG wire#powerrail
      Contact( "ZSC-21.11" )
   END_RUNG wire#w3
   RUNG wire#powerrail
      I_Contact( #"AV-21.11".QCMD_OP )
   END_RUNG wire#w3
   // the same network as SCL:
   #"AV-21.11"(LOCK := #lock,   // "Valve"
               LIOP_SEL := #Init,
               L_AUT := #Init,
               L_REMOTE := #Init,
               L_RESET := #Reset,
               AUT_OP := ("T-21.00_DB".ChiliAwet_3.V_CMD AND "T-04.01_DB".Actuator.AV_Outlet) OR ("T-04.01_DB".Cmd.Flushing AND "T-04.01_DB".State.Flush_selected.%X1),
               FB_OPEN := NOT "ZSC-21.11" AND #"AV-21.11".QCMD_OP,
               FB_CLOSE := "ZSC-21.11" OR NOT #"AV-21.11".QCMD_OP,
               L_MON := #Init,
               INSTANCE := 'AV-21.11',
               QCMD_OP => "AV-21.11");
END_REGION

REGION Network 40: AV-21.12
